LIN {X 0.200,Y -475.313,Z 1141.533,A 0.000,B 0.000,C 90.000,E1 275.853} C_DIS
LIN {X -0.137,Y -474.500,Z 1141.530,A 0.000,B 0.000,C 90.000,E1 275.391} C_DIS
LIN {X -0.046,Y -473.245,Z 1141.527,A 0.000,B 0.000,C 90.000,E1 274.878} C_DIS
LIN {X 0.081,Y -471.579,Z 1141.524,A 0.000,B 0.000,C 90.000,E1 274.359} C_DIS
LIN {X 0.199,Y -469.321,Z 1141.521,A 0.000,B 0.000,C 90.000,E1 273.841} C_DIS
LIN {X 0.000,Y -468.016,Z 1141.520,A 0.000,B 0.000,C 90.000,E1 273.612} C_DIS
LIN {X 0.090,Y -464.739,Z 1141.517,A 0.000,B 0.000,C 90.000,E1 273.094} C_DIS
LIN {X -0.113,Y -462.816,Z 1141.516,A 0.000,B 0.000,C 90.000,E1 272.865} C_DIS
LIN {X -0.071,Y -458.078,Z 1141.513,A 0.000,B 0.000,C 90.000,E1 272.350} C_DIS
LIN {X 0.192,Y -455.207,Z 1141.512,A 0.000,B 0.000,C 90.000,E1 272.064} C_DIS
LIN {X 0.157,Y -448.955,Z 1141.509,A 0.000,B 0.000,C 90.000,E1 271.604} C_DIS
LIN {X -0.185,Y -442.338,Z 1141.507,A 0.000,B 0.000,C 90.000,E1 271.260} C_DIS
LIN {X -0.038,Y -435.436,Z 1141.505,A 0.000,B 0.000,C 90.000,E1 270.917} C_DIS
LIN {X 0.066,Y -428.431,Z 1141.504,A 0.000,B 0.000,C 90.000,E1 270.630} C_DIS
LIN {X 0.073,Y -421.301,Z 1141.502,A 0.000,B 0.000,C 90.000,E1 270.401} C_DIS
LIN {X -0.072,Y -414.046,Z 1141.501,A 0.000,B 0.000,C 90.000,E1 270.229} C_DIS
LIN {X -0.082,Y -402.883,Z 1141.500,A 0.000,B 0.000,C 90.000,E1 270.000} C_DIS
LIN {X -0.091,Y -391.480,Z 1141.499,A 0.000,B 0.000,C 90.000,E1 269.828} C_DIS
LIN {X -0.150,Y -380.857,Z 1141.499,A 0.000,B 0.000,C 90.000,E1 269.771} C_DIS
LIN {X 0.176,Y -377.810,Z 1141.499,A 0.000,B 0.000,C 90.000,E1 269.714} C_DIS
LIN {X 0.059,Y -181.500,Z 1141.499,A 0.000,B 0.000,C 90.000,E1 269.714} C_DIS
LIN {X 0.062,Y -180.907,Z 1141.475,A 0.000,B 0.000,C 90.000,E1 265.469} C_DIS
LIN {X -0.062,Y -180.745,Z 1141.470,A 0.000,B 0.000,C 90.000,E1 264.666} C_DIS
LIN {X 0.007,Y -178.837,Z 1141.442,A 0.000,B 0.000,C 90.000,E1 259.577} C_DIS
LIN {X -0.096,Y -175.880,Z 1141.414,A 0.000,B 0.000,C 90.000,E1 254.519} C_DIS
LIN {X 0.010,Y -174.542,Z 1141.404,A 0.000,B 0.000,C 90.000,E1 252.779} C_DIS
LIN {X 0.103,Y -171.527,Z 1141.380,A 0.000,B 0.000,C 90.000,E1 248.465} C_DIS
LIN {X 0.089,Y -167.753,Z 1141.357,A 0.000,B 0.000,C 90.000,E1 244.152} C_DIS
LIN {X 0.026,Y -166.456,Z 1141.347,A 0.000,B 0.000,C 90.000,E1 242.436} C_DIS
LIN {X 0.017,Y -163.172,Z 1141.328,A 0.000,B 0.000,C 90.000,E1 238.948} C_DIS
LIN {X 0.066,Y -161.131,Z 1141.313,A 0.000,B 0.000,C 90.000,E1 236.294} C_DIS
LIN {X -0.032,Y -157.153,Z 1141.288,A 0.000,B 0.000,C 90.000,E1 231.904} C_DIS
LIN {X -0.009,Y -155.885,Z 1141.278,A 0.000,B 0.000,C 90.000,E1 230.114} C_DIS
LIN {X -0.050,Y -152.135,Z 1141.254,A 0.000,B 0.000,C 90.000,E1 225.648} C_DIS
LIN {X -0.030,Y -150.385,Z 1141.238,A 0.000,B 0.000,C 90.000,E1 222.933} C_DIS
LIN {X -0.005,Y -147.117,Z 1141.213,A 0.000,B 0.000,C 90.000,E1 218.382} C_DIS
LIN {X -0.015,Y -145.682,Z 1141.198,A 0.000,B 0.000,C 90.000,E1 215.644} C_DIS
LIN {X -0.017,Y -143.065,Z 1141.172,A 0.000,B 0.000,C 90.000,E1 211.052} C_DIS
LIN {X 0.041,Y -141.686,Z 1141.152,A 0.000,B 0.000,C 90.000,E1 207.334} C_DIS
LIN {X 0.019,Y -139.459,Z 1141.116,A 0.000,B 0.000,C 90.000,E1 200.844} C_DIS
LIN {X 0.069,Y -139.193,Z 1141.105,A 0.000,B 0.000,C 90.000,E1 198.960} C_DIS
LIN {X -0.044,Y -138.325,Z 1141.054,A 0.000,B 0.000,C 90.000,E1 189.670} C_DIS
LIN {X -0.039,Y -139.453,Z 1141.007,A 0.000,B 0.000,C 90.000,E1 181.260} C_DIS
LIN {X 0.041,Y -141.000,Z 1140.976,A 0.000,B 0.000,C 90.000,E1 175.641} C_DIS
LIN {X -0.009,Y -142.755,Z 1140.955,A 0.000,B 0.000,C 90.000,E1 171.951} C_DIS
LIN {X -0.054,Y -145.157,Z 1140.930,A 0.000,B 0.000,C 90.000,E1 167.353} C_DIS
LIN {X -0.061,Y -147.779,Z 1140.909,A 0.000,B 0.000,C 90.000,E1 163.685} C_DIS
LIN {X 0.019,Y -150.457,Z 1140.889,A 0.000,B 0.000,C 90.000,E1 160.007} C_DIS
LIN {X -0.048,Y -153.906,Z 1140.869,A 0.000,B 0.000,C 90.000,E1 156.410} C_DIS
LIN {X 0.017,Y -157.316,Z 1140.849,A 0.000,B 0.000,C 90.000,E1 152.794} C_DIS
LIN {X -0.036,Y -161.504,Z 1140.829,A 0.000,B 0.000,C 90.000,E1 149.253} C_DIS
LIN {X -0.020,Y -165.703,Z 1140.810,A 0.000,B 0.000,C 90.000,E1 145.722} C_DIS
LIN {X 0.106,Y -170.649,Z 1140.790,A 0.000,B 0.000,C 90.000,E1 142.190} C_DIS
LIN {X 0.018,Y -175.524,Z 1140.771,A 0.000,B 0.000,C 90.000,E1 138.771} C_DIS
LIN {X 0.012,Y -181.144,Z 1140.752,A 0.000,B 0.000,C 90.000,E1 135.364} C_DIS
LIN {X 0.010,Y -186.596,Z 1140.733,A 0.000,B 0.000,C 90.000,E1 132.000} C_DIS
LIN {X 0.080,Y -191.206,Z 1140.719,A 0.000,B 0.000,C 90.000,E1 129.483} C_DIS
LIN {X 0.004,Y -197.018,Z 1140.701,A 0.000,B 0.000,C 90.000,E1 126.217} C_DIS
LIN {X -0.072,Y -201.191,Z 1140.689,A 0.000,B 0.000,C 90.000,E1 124.119} C_DIS
LIN {X 0.092,Y -310.929,Z 1140.689,A 0.000,B 0.000,C 90.000,E1 124.072} C_DIS
LIN {X 0.092,Y -315.579,Z 1140.688,A 0.000,B 0.000,C 90.000,E1 123.913} C_DIS
LIN {X -0.033,Y -317.772,Z 1140.688,A 0.000,B 0.000,C 90.000,E1 123.785} C_DIS
LIN {X -0.005,Y -321.647,Z 1140.685,A 0.000,B 0.000,C 90.000,E1 123.372} C_DIS
LIN {X -0.032,Y -323.552,Z 1140.684,A 0.000,B 0.000,C 90.000,E1 123.086} C_DIS
LIN {X -0.060,Y -325.048,Z 1140.682,A 0.000,B 0.000,C 90.000,E1 122.801} C_DIS
LIN {X -0.046,Y -328.621,Z 1140.677,A 0.000,B 0.000,C 90.000,E1 121.848} C_DIS
LIN {X -0.027,Y -339.698,Z 1140.661,A 0.000,B 0.000,C 90.000,E1 119.027} C_DIS
LIN {X 0.170,Y -352.167,Z 1140.646,A 0.000,B 0.000,C 90.000,E1 116.232} C_DIS
LIN {X -0.081,Y -366.144,Z 1140.631,A 0.000,B 0.000,C 90.000,E1 113.567} C_DIS
LIN {X -0.161,Y -379.928,Z 1140.618,A 0.000,B 0.000,C 90.000,E1 111.227} C_DIS
LIN {X -0.023,Y -395.095,Z 1140.605,A 0.000,B 0.000,C 90.000,E1 108.906} C_DIS
LIN {X -0.141,Y -411.753,Z 1140.593,A 0.000,B 0.000,C 90.000,E1 106.677} C_DIS
LIN {X -0.085,Y -430.020,Z 1140.580,A 0.000,B 0.000,C 90.000,E1 104.481} C_DIS
LIN {X 0.106,Y -449.754,Z 1140.569,A 0.000,B 0.000,C 90.000,E1 102.355} C_DIS
LIN {X 0.080,Y -467.535,Z 1140.559,A 0.000,B 0.000,C 90.000,E1 100.658} C_DIS
LIN {X 0.008,Y -469.919,Z 1140.558,A 0.000,B 0.000,C 90.000,E1 100.433} C_DIS
LIN {X -0.067,Y -471.794,Z 1140.557,A 0.000,B 0.000,C 90.000,E1 100.197} C_DIS
LIN {X -0.143,Y -473.215,Z 1140.555,A 0.000,B 0.000,C 90.000,E1 99.962} C_DIS
LIN {X -0.037,Y -475.103,Z 1140.552,A 0.000,B 0.000,C 90.000,E1 99.443} C_DIS
LIN {X 0.157,Y -475.883,Z 1140.550,A 0.000,B 0.000,C 90.000,E1 98.916} C_DIS
LIN {X -0.184,Y -475.689,Z 1140.547,A 0.000,B 0.000,C 90.000,E1 98.454} C_DIS
LIN {X -0.047,Y -474.497,Z 1140.544,A 0.000,B 0.000,C 90.000,E1 97.936} C_DIS
LIN {X -0.182,Y -473.472,Z 1140.543,A 0.000,B 0.000,C 90.000,E1 97.701} C_DIS
LIN {X 0.151,Y -472.094,Z 1140.541,A 0.000,B 0.000,C 90.000,E1 97.409} C_DIS
LIN {X 0.048,Y -457.591,Z 1140.530,A 0.000,B 0.000,C 90.000,E1 95.391} C_DIS
LIN {X 0.126,Y -438.390,Z 1140.514,A 0.000,B 0.000,C 90.000,E1 92.522} C_DIS
LIN {X 0.138,Y -419.215,Z 1140.496,A 0.000,B 0.000,C 90.000,E1 89.312} C_DIS
LIN {X -0.010,Y -408.971,Z 1140.486,A 0.000,B 0.000,C 90.000,E1 87.421} C_DIS
LIN {X 0.054,Y -398.485,Z 1140.475,A 0.000,B 0.000,C 90.000,E1 85.469} C_DIS
LIN {X 0.018,Y -385.098,Z 1140.461,A 0.000,B 0.000,C 90.000,E1 82.932} C_DIS
LIN {X 0.082,Y -376.107,Z 1140.451,A 0.000,B 0.000,C 90.000,E1 81.197} C_DIS
LIN {X 0.036,Y -366.859,Z 1140.441,A 0.000,B 0.000,C 90.000,E1 79.454} C_DIS
LIN {X -0.074,Y -358.902,Z 1140.433,A 0.000,B 0.000,C 90.000,E1 77.993} C_DIS
LIN {X -0.002,Y -347.398,Z 1140.422,A 0.000,B 0.000,C 90.000,E1 75.880} C_DIS
LIN {X -0.026,Y -334.287,Z 1140.408,A 0.000,B 0.000,C 90.000,E1 73.433} C_DIS
LIN {X -0.001,Y -320.080,Z 1140.392,A 0.000,B 0.000,C 90.000,E1 70.604} C_DIS
LIN {X 0.053,Y -303.837,Z 1140.373,A 0.000,B 0.000,C 90.000,E1 67.050} C_DIS
LIN {X 0.038,Y -291.318,Z 1140.356,A 0.000,B 0.000,C 90.000,E1 64.076} C_DIS
LIN {X -0.058,Y -279.221,Z 1140.339,A 0.000,B 0.000,C 90.000,E1 61.051} C_DIS
LIN {X 0.049,Y -267.755,Z 1140.322,A 0.000,B 0.000,C 90.000,E1 57.916} C_DIS
LIN {X -0.102,Y -256.802,Z 1140.304,A 0.000,B 0.000,C 90.000,E1 54.769} C_DIS
LIN {X 0.031,Y -245.381,Z 1140.284,A 0.000,B 0.000,C 90.000,E1 51.126} C_DIS
LIN {X -0.112,Y -235.027,Z 1140.264,A 0.000,B 0.000,C 90.000,E1 47.472} C_DIS
LIN {X 0.030,Y -227.285,Z 1140.247,A 0.000,B 0.000,C 90.000,E1 44.433} C_DIS
LIN {X -0.012,Y -218.155,Z 1140.226,A 0.000,B 0.000,C 90.000,E1 40.620} C_DIS
LIN {X -0.066,Y -211.276,Z 1140.208,A 0.000,B 0.000,C 90.000,E1 37.523} C_DIS
LIN {X 0.079,Y -204.769,Z 1140.191,A 0.000,B 0.000,C 90.000,E1 34.326} C_DIS
LIN {X 0.015,Y -197.461,Z 1140.169,A 0.000,B 0.000,C 90.000,E1 30.335} C_DIS
LIN {X 0.028,Y -192.220,Z 1140.151,A 0.000,B 0.000,C 90.000,E1 27.078} C_DIS
LIN {X 0.055,Y -186.581,Z 1140.128,A 0.000,B 0.000,C 90.000,E1 22.950} C_DIS
LIN {X 0.058,Y -181.865,Z 1140.104,A 0.000,B 0.000,C 90.000,E1 18.779} C_DIS
LIN {X -0.023,Y -178.162,Z 1140.081,A 0.000,B 0.000,C 90.000,E1 14.592} C_DIS
LIN {X -0.047,Y -175.079,Z 1140.053,A 0.000,B 0.000,C 90.000,E1 9.500} C_DIS
LIN {X 0.015,Y -173.270,Z 1140.005,A 0.000,B 0.000,C 90.000,E1 0.917} C_DIS
LIN {X 0.050,Y -174.989,Z 1139.964,A 0.000,B 0.000,C 90.000,E1 353.514} C_DIS
LIN {X 0.006,Y -177.963,Z 1139.936,A 0.000,B 0.000,C 90.000,E1 348.409} C_DIS
LIN {X 0.056,Y -181.448,Z 1139.912,A 0.000,B 0.000,C 90.000,E1 344.157} C_DIS
LIN {X -0.110,Y -185.852,Z 1139.889,A 0.000,B 0.000,C 90.000,E1 340.007} C_DIS
LIN {X 0.074,Y -191.032,Z 1139.866,A 0.000,B 0.000,C 90.000,E1 335.793} C_DIS
LIN {X -0.045,Y -195.878,Z 1139.847,A 0.000,B 0.000,C 90.000,E1 332.538} C_DIS
LIN {X -0.043,Y -201.277,Z 1139.829,A 0.000,B 0.000,C 90.000,E1 329.282} C_DIS
LIN {X -0.121,Y -207.264,Z 1139.811,A 0.000,B 0.000,C 90.000,E1 326.087} C_DIS
LIN {X -0.032,Y -214.122,Z 1139.794,A 0.000,B 0.000,C 90.000,E1 322.889} C_DIS
LIN {X -0.049,Y -222.780,Z 1139.774,A 0.000,B 0.000,C 90.000,E1 319.380} C_DIS
LIN {X 0.034,Y -231.481,Z 1139.757,A 0.000,B 0.000,C 90.000,E1 316.296} C_DIS
LIN {X 0.001,Y -241.200,Z 1139.741,A 0.000,B 0.000,C 90.000,E1 313.299} C_DIS
LIN {X -0.106,Y -252.087,Z 1139.724,A 0.000,B 0.000,C 90.000,E1 310.378} C_DIS
LIN {X 0.139,Y -264.307,Z 1139.708,A 0.000,B 0.000,C 90.000,E1 307.443} C_DIS
LIN {X -0.053,Y -279.632,Z 1139.691,A 0.000,B 0.000,C 90.000,E1 304.326} C_DIS
LIN {X -0.018,Y -292.655,Z 1139.677,A 0.000,B 0.000,C 90.000,E1 301.926} C_DIS
LIN {X -0.124,Y -308.904,Z 1139.663,A 0.000,B 0.000,C 90.000,E1 299.283} C_DIS
LIN {X 0.042,Y -326.808,Z 1139.648,A 0.000,B 0.000,C 90.000,E1 296.668} C_DIS
LIN {X 0.124,Y -341.553,Z 1139.638,A 0.000,B 0.000,C 90.000,E1 294.771} C_DIS
LIN {X 0.091,Y -354.713,Z 1139.629,A 0.000,B 0.000,C 90.000,E1 293.259} C_DIS
LIN {X 0.010,Y -368.110,Z 1139.622,A 0.000,B 0.000,C 90.000,E1 291.897} C_DIS
LIN {X -0.061,Y -392.786,Z 1139.609,A 0.000,B 0.000,C 90.000,E1 289.631} C_DIS
LIN {X -0.033,Y -403.534,Z 1139.604,A 0.000,B 0.000,C 90.000,E1 288.652} C_DIS
LIN {X 0.210,Y -411.431,Z 1139.599,A 0.000,B 0.000,C 90.000,E1 287.873} C_DIS
LIN {X 0.215,Y -421.680,Z 1139.594,A 0.000,B 0.000,C 90.000,E1 286.858} C_DIS
LIN {X 0.218,Y -429.215,Z 1139.589,A 0.000,B 0.000,C 90.000,E1 286.079} C_DIS
LIN {X 0.086,Y -436.426,Z 1139.585,A 0.000,B 0.000,C 90.000,E1 285.300} C_DIS
LIN {X -0.180,Y -443.169,Z 1139.581,A 0.000,B 0.000,C 90.000,E1 284.537} C_DIS
LIN {X 0.056,Y -449.195,Z 1139.576,A 0.000,B 0.000,C 90.000,E1 283.716} C_DIS
LIN {X 0.011,Y -454.502,Z 1139.572,A 0.000,B 0.000,C 90.000,E1 282.939} C_DIS
LIN {X -0.091,Y -459.121,Z 1139.568,A 0.000,B 0.000,C 90.000,E1 282.175} C_DIS
LIN {X -0.252,Y -463.156,Z 1139.563,A 0.000,B 0.000,C 90.000,E1 281.422} C_DIS
LIN {X 0.020,Y -467.739,Z 1139.558,A 0.000,B 0.000,C 90.000,E1 280.366} C_DIS
LIN {X 0.093,Y -469.729,Z 1139.555,A 0.000,B 0.000,C 90.000,E1 279.849} C_DIS
LIN {X -0.209,Y -471.485,Z 1139.552,A 0.000,B 0.000,C 90.000,E1 279.378} C_DIS
LIN {X -0.115,Y -473.007,Z 1139.549,A 0.000,B 0.000,C 90.000,E1 278.859} C_DIS
LIN {X -0.005,Y -474.223,Z 1139.546,A 0.000,B 0.000,C 90.000,E1 278.341} C_DIS
LIN {X 0.180,Y -475.168,Z 1139.544,A 0.000,B 0.000,C 90.000,E1 277.814} C_DIS
LIN {X -0.164,Y -475.768,Z 1139.541,A 0.000,B 0.000,C 90.000,E1 277.352} C_DIS
LIN {X -0.032,Y -476.050,Z 1139.538,A 0.000,B 0.000,C 90.000,E1 276.834} C_DIS
LIN {X 0.105,Y -475.977,Z 1139.535,A 0.000,B 0.000,C 90.000,E1 276.315} C_DIS
LIN {X 0.243,Y -475.515,Z 1139.532,A 0.000,B 0.000,C 90.000,E1 275.796} C_DIS
LIN {X -0.094,Y -474.683,Z 1139.530,A 0.000,B 0.000,C 90.000,E1 275.334} C_DIS
LIN {X -0.002,Y -473.432,Z 1139.527,A 0.000,B 0.000,C 90.000,E1 274.821} C_DIS
LIN {X 0.128,Y -471.721,Z 1139.524,A 0.000,B 0.000,C 90.000,E1 274.302} C_DIS
LIN {X -0.223,Y -469.455,Z 1139.521,A 0.000,B 0.000,C 90.000,E1 273.841} C_DIS
LIN {X -0.150,Y -466.592,Z 1139.518,A 0.000,B 0.000,C 90.000,E1 273.326} C_DIS
LIN {X -0.065,Y -462.911,Z 1139.516,A 0.000,B 0.000,C 90.000,E1 272.808} C_DIS
LIN {X -0.023,Y -458.133,Z 1139.513,A 0.000,B 0.000,C 90.000,E1 272.293} C_DIS
LIN {X -0.206,Y -455.209,Z 1139.511,A 0.000,B 0.000,C 90.000,E1 272.064} C_DIS
LIN {X -0.213,Y -448.901,Z 1139.509,A 0.000,B 0.000,C 90.000,E1 271.604} C_DIS
LIN {X -0.091,Y -442.192,Z 1139.507,A 0.000,B 0.000,C 90.000,E1 271.203} C_DIS
LIN {X 0.068,Y -435.279,Z 1139.505,A 0.000,B 0.000,C 90.000,E1 270.859} C_DIS
LIN {X 0.194,Y -428.312,Z 1139.503,A 0.000,B 0.000,C 90.000,E1 270.573} C_DIS
LIN {X -0.207,Y -421.182,Z 1139.502,A 0.000,B 0.000,C 90.000,E1 270.401} C_DIS
LIN {X 0.081,Y -413.850,Z 1139.501,A 0.000,B 0.000,C 90.000,E1 270.172} C_DIS
LIN {X 0.084,Y -402.501,Z 1139.500,A 0.000,B 0.000,C 90.000,E1 269.943} C_DIS
LIN {X 0.059,Y -394.923,Z 1139.499,A 0.000,B 0.000,C 90.000,E1 269.828} C_DIS
LIN {X -0.055,Y -388.034,Z 1139.499,A 0.000,B 0.000,C 90.000,E1 269.771} C_DIS
LIN {X 0.056,Y -378.077,Z 1139.498,A 0.000,B 0.000,C 90.000,E1 269.714} C_DIS
LIN {X 0.001,Y -181.494,Z 1139.498,A 0.000,B 0.000,C 90.000,E1 269.714} C_DIS
LIN {X -0.020,Y -180.907,Z 1139.475,A 0.000,B 0.000,C 90.000,E1 265.469} C_DIS
LIN {X 0.037,Y -180.733,Z 1139.470,A 0.000,B 0.000,C 90.000,E1 264.609} C_DIS
LIN {X -0.042,Y -178.823,Z 1139.442,A 0.000,B 0.000,C 90.000,E1 259.567} C_DIS
LIN {X 0.040,Y -175.868,Z 1139.414,A 0.000,B 0.000,C 90.000,E1 254.448} C_DIS
LIN {X 0.034,Y -173.838,Z 1139.399,A 0.000,B 0.000,C 90.000,E1 251.891} C_DIS
LIN {X 0.023,Y -171.505,Z 1139.380,A 0.000,B 0.000,C 90.000,E1 248.465} C_DIS
LIN {X 0.010,Y -167.733,Z 1139.356,A 0.000,B 0.000,C 90.000,E1 244.152} C_DIS
LIN {X 0.026,Y -166.430,Z 1139.347,A 0.000,B 0.000,C 90.000,E1 242.410} C_DIS
LIN {X -0.060,Y -163.150,Z 1139.327,A 0.000,B 0.000,C 90.000,E1 238.948} C_DIS
LIN {X -0.011,Y -161.105,Z 1139.313,A 0.000,B 0.000,C 90.000,E1 236.294} C_DIS
LIN {X -0.027,Y -157.833,Z 1139.293,A 0.000,B 0.000,C 90.000,E1 232.763} C_DIS
LIN {X 0.036,Y -155.865,Z 1139.278,A 0.000,B 0.000,C 90.000,E1 230.070} C_DIS
LIN {X 0.091,Y -152.115,Z 1139.253,A 0.000,B 0.000,C 90.000,E1 225.567} C_DIS
LIN {X -0.001,Y -150.366,Z 1139.238,A 0.000,B 0.000,C 90.000,E1 222.894} C_DIS
LIN {X 0.038,Y -147.101,Z 1139.213,A 0.000,B 0.000,C 90.000,E1 218.338} C_DIS
LIN {X 0.031,Y -145.669,Z 1139.198,A 0.000,B 0.000,C 90.000,E1 215.598} C_DIS
LIN {X 0.035,Y -143.051,Z 1139.172,A 0.000,B 0.000,C 90.000,E1 211.003} C_DIS
LIN {X -0.030,Y -141.674,Z 1139.152,A 0.000,B 0.000,C 90.000,E1 207.334} C_DIS
LIN {X 0.079,Y -139.454,Z 1139.116,A 0.000,B 0.000,C 90.000,E1 200.791} C_DIS
LIN {X 0.000,Y -139.188,Z 1139.105,A 0.000,B 0.000,C 90.000,E1 198.960} C_DIS
LIN {X 0.023,Y -138.323,Z 1139.053,A 0.000,B 0.000,C 90.000,E1 189.613} C_DIS
LIN {X 0.030,Y -139.458,Z 1139.007,A 0.000,B 0.000,C 90.000,E1 181.203} C_DIS
LIN {X -0.029,Y -141.012,Z 1138.976,A 0.000,B 0.000,C 90.000,E1 175.641} C_DIS
LIN {X 0.061,Y -142.766,Z 1138.955,A 0.000,B 0.000,C 90.000,E1 171.894} C_DIS
LIN {X 0.016,Y -145.175,Z 1138.929,A 0.000,B 0.000,C 90.000,E1 167.297} C_DIS
LIN {X 0.050,Y -147.796,Z 1138.909,A 0.000,B 0.000,C 90.000,E1 163.614} C_DIS
LIN {X -0.055,Y -150.480,Z 1138.889,A 0.000,B 0.000,C 90.000,E1 160.007} C_DIS
LIN {X 0.019,Y -153.935,Z 1138.869,A 0.000,B 0.000,C 90.000,E1 156.357} C_DIS
LIN {X 0.082,Y -157.346,Z 1138.849,A 0.000,B 0.000,C 90.000,E1 152.743} C_DIS
LIN {X 0.026,Y -161.540,Z 1138.829,A 0.000,B 0.000,C 90.000,E1 149.203} C_DIS
LIN {X 0.039,Y -165.738,Z 1138.809,A 0.000,B 0.000,C 90.000,E1 145.674} C_DIS
LIN {X 0.026,Y -170.691,Z 1138.790,A 0.000,B 0.000,C 90.000,E1 142.190} C_DIS
LIN {X -0.062,Y -175.564,Z 1138.771,A 0.000,B 0.000,C 90.000,E1 138.771} C_DIS
LIN {X 0.057,Y -181.182,Z 1138.752,A 0.000,B 0.000,C 90.000,E1 135.324} C_DIS
LIN {X -0.074,Y -186.642,Z 1138.733,A 0.000,B 0.000,C 90.000,E1 132.000} C_DIS
LIN {X -0.005,Y -191.248,Z 1138.719,A 0.000,B 0.000,C 90.000,E1 129.483} C_DIS
LIN {X -0.082,Y -197.066,Z 1138.701,A 0.000,B 0.000,C 90.000,E1 126.217} C_DIS
LIN {X -0.010,Y -201.161,Z 1138.690,A 0.000,B 0.000,C 90.000,E1 124.119} C_DIS
LIN {X -0.074,Y -310.690,Z 1138.689,A 0.000,B 0.000,C 90.000,E1 124.119} C_DIS
LIN {X 0.066,Y -315.833,Z 1138.688,A 0.000,B 0.000,C 90.000,E1 123.913} C_DIS
LIN {X -0.171,Y -318.170,Z 1138.688,A 0.000,B 0.000,C 90.000,E1 123.785} C_DIS
LIN {X 0.172,Y -322.022,Z 1138.685,A 0.000,B 0.000,C 90.000,E1 123.293} C_DIS
LIN {X -0.104,Y -323.897,Z 1138.683,A 0.000,B 0.000,C 90.000,E1 123.038} C_DIS
LIN {X 0.068,Y -325.366,Z 1138.682,A 0.000,B 0.000,C 90.000,E1 122.704} C_DIS
LIN {X -0.132,Y -338.678,Z 1138.663,A 0.000,B 0.000,C 90.000,E1 119.283} C_DIS
LIN {X 0.025,Y -351.027,Z 1138.647,A 0.000,B 0.000,C 90.000,E1 116.488} C_DIS
LIN {X 0.078,Y -364.867,Z 1138.632,A 0.000,B 0.000,C 90.000,E1 113.770} C_DIS
LIN {X 0.120,Y -378.524,Z 1138.619,A 0.000,B 0.000,C 90.000,E1 111.408} C_DIS
LIN {X -0.140,Y -393.553,Z 1138.606,A 0.000,B 0.000,C 90.000,E1 109.141} C_DIS
LIN {X 0.087,Y -410.062,Z 1138.594,A 0.000,B 0.000,C 90.000,E1 106.858} C_DIS
LIN {X 0.112,Y -428.168,Z 1138.582,A 0.000,B 0.000,C 90.000,E1 104.662} C_DIS
LIN {X -0.214,Y -447.792,Z 1138.570,A 0.000,B 0.000,C 90.000,E1 102.591} C_DIS
LIN {X 0.091,Y -468.110,Z 1138.559,A 0.000,B 0.000,C 90.000,E1 100.602} C_DIS
LIN {X 0.110,Y -470.350,Z 1138.558,A 0.000,B 0.000,C 90.000,E1 100.366} C_DIS
LIN {X -0.122,Y -472.163,Z 1138.556,A 0.000,B 0.000,C 90.000,E1 100.141} C_DIS
LIN {X 0.196,Y -473.524,Z 1138.555,A 0.000,B 0.000,C 90.000,E1 99.849} C_DIS
LIN {X -0.084,Y -475.233,Z 1138.552,A 0.000,B 0.000,C 90.000,E1 99.378} C_DIS
LIN {X 0.034,Y -475.869,Z 1138.549,A 0.000,B 0.000,C 90.000,E1 98.859} C_DIS
LIN {X 0.167,Y -475.536,Z 1138.547,A 0.000,B 0.000,C 90.000,E1 98.341} C_DIS
LIN {X -0.102,Y -474.189,Z 1138.544,A 0.000,B 0.000,C 90.000,E1 97.871} C_DIS
LIN {X 0.168,Y -473.070,Z 1138.542,A 0.000,B 0.000,C 90.000,E1 97.587} C_DIS
LIN {X 0.030,Y -471.574,Z 1138.541,A 0.000,B 0.000,C 90.000,E1 97.352} C_DIS
LIN {X 0.145,Y -455.223,Z 1138.528,A 0.000,B 0.000,C 90.000,E1 95.049} C_DIS
LIN {X -0.183,Y -439.529,Z 1138.515,A 0.000,B 0.000,C 90.000,E1 92.751} C_DIS
LIN {X 0.178,Y -421.764,Z 1138.499,A 0.000,B 0.000,C 90.000,E1 89.771} C_DIS
LIN {X -0.165,Y -408.479,Z 1138.485,A 0.000,B 0.000,C 90.000,E1 87.364} C_DIS
LIN {X -0.108,Y -397.980,Z 1138.474,A 0.000,B 0.000,C 90.000,E1 85.412} C_DIS
LIN {X -0.153,Y -384.603,Z 1138.460,A 0.000,B 0.000,C 90.000,E1 82.875} C_DIS
LIN {X -0.096,Y -375.592,Z 1138.451,A 0.000,B 0.000,C 90.000,E1 81.141} C_DIS
LIN {X -0.148,Y -366.316,Z 1138.441,A 0.000,B 0.000,C 90.000,E1 79.398} C_DIS
LIN {X 0.086,Y -358.335,Z 1138.433,A 0.000,B 0.000,C 90.000,E1 77.881} C_DIS
LIN {X -0.117,Y -346.817,Z 1138.421,A 0.000,B 0.000,C 90.000,E1 75.811} C_DIS
LIN {X 0.085,Y -333.720,Z 1138.407,A 0.000,B 0.000,C 90.000,E1 73.323} C_DIS
LIN {X 0.080,Y -319.500,Z 1138.392,A 0.000,B 0.000,C 90.000,E1 70.496} C_DIS
LIN {X -0.063,Y -303.309,Z 1138.372,A 0.000,B 0.000,C 90.000,E1 66.975} C_DIS
LIN {X 0.053,Y -290.796,Z 1138.355,A 0.000,B 0.000,C 90.000,E1 63.973} C_DIS
LIN {X 0.066,Y -278.715,Z 1138.339,A 0.000,B 0.000,C 90.000,E1 60.923} C_DIS
LIN {X 0.151,Y -267.269,Z 1138.321,A 0.000,B 0.000,C 90.000,E1 57.788} C_DIS
LIN {X -0.021,Y -256.318,Z 1138.304,A 0.000,B 0.000,C 90.000,E1 54.642} C_DIS
LIN {X 0.041,Y -245.979,Z 1138.286,A 0.000,B 0.000,C 90.000,E1 51.376} C_DIS
LIN {X -0.032,Y -236.536,Z 1138.267,A 0.000,B 0.000,C 90.000,E1 48.081} C_DIS
LIN {X -0.012,Y -228.708,Z 1138.250,A 0.000,B 0.000,C 90.000,E1 45.081} C_DIS
LIN {X -0.025,Y -219.457,Z 1138.229,A 0.000,B 0.000,C 90.000,E1 41.272} C_DIS
LIN {X -0.052,Y -212.462,Z 1138.212,A 0.000,B 0.000,C 90.000,E1 38.177} C_DIS
LIN {X 0.071,Y -204.260,Z 1138.190,A 0.000,B 0.000,C 90.000,E1 34.199} C_DIS
LIN {X -0.004,Y -196.963,Z 1138.168,A 0.000,B 0.000,C 90.000,E1 30.207} C_DIS
LIN {X -0.002,Y -191.740,Z 1138.150,A 0.000,B 0.000,C 90.000,E1 26.950} C_DIS
LIN {X 0.011,Y -186.124,Z 1138.127,A 0.000,B 0.000,C 90.000,E1 22.823} C_DIS
LIN {X -0.059,Y -181.433,Z 1138.104,A 0.000,B 0.000,C 90.000,E1 18.671} C_DIS
LIN {X 0.029,Y -177.741,Z 1138.080,A 0.000,B 0.000,C 90.000,E1 14.426} C_DIS
LIN {X 0.027,Y -174.715,Z 1138.052,A 0.000,B 0.000,C 90.000,E1 9.321} C_DIS
LIN {X 0.000,Y -173.011,Z 1138.000,A 0.000,B 0.000,C 90.000,E1 360.000} C_DIS
LIN {X 0.071,Y -175.091,Z 1137.959,A 0.000,B 0.000,C 90.000,E1 352.648} C_DIS
LIN {X 0.100,Y -178.266,Z 1137.931,A 0.000,B 0.000,C 90.000,E1 347.521} C_DIS
LIN {X -0.011,Y -181.920,Z 1137.907,A 0.000,B 0.000,C 90.000,E1 343.323} C_DIS
LIN {X -0.041,Y -186.439,Z 1137.884,A 0.000,B 0.000,C 90.000,E1 339.135} C_DIS
LIN {X -0.007,Y -191.815,Z 1137.861,A 0.000,B 0.000,C 90.000,E1 334.973} C_DIS
LIN {X -0.019,Y -196.817,Z 1137.843,A 0.000,B 0.000,C 90.000,E1 331.691} C_DIS
LIN {X -0.064,Y -202.409,Z 1137.825,A 0.000,B 0.000,C 90.000,E1 328.456} C_DIS
LIN {X 0.006,Y -208.616,Z 1137.807,A 0.000,B 0.000,C 90.000,E1 325.229} C_DIS
LIN {X 0.008,Y -215.710,Z 1137.789,A 0.000,B 0.000,C 90.000,E1 322.065} C_DIS
LIN {X 0.079,Y -223.587,Z 1137.772,A 0.000,B 0.000,C 90.000,E1 318.933} C_DIS
LIN {X 0.018,Y -232.452,Z 1137.755,A 0.000,B 0.000,C 90.000,E1 315.891} C_DIS
LIN {X 0.010,Y -242.342,Z 1137.738,A 0.000,B 0.000,C 90.000,E1 312.894} C_DIS
LIN {X 0.123,Y -253.399,Z 1137.722,A 0.000,B 0.000,C 90.000,E1 309.930} C_DIS
LIN {X 0.041,Y -265.853,Z 1137.706,A 0.000,B 0.000,C 90.000,E1 307.076} C_DIS
LIN {X 0.124,Y -281.426,Z 1137.689,A 0.000,B 0.000,C 90.000,E1 303.913} C_DIS
LIN {X 0.044,Y -296.633,Z 1137.673,A 0.000,B 0.000,C 90.000,E1 301.209} C_DIS
LIN {X 0.006,Y -311.175,Z 1137.661,A 0.000,B 0.000,C 90.000,E1 298.899} C_DIS
LIN {X 0.095,Y -329.306,Z 1137.646,A 0.000,B 0.000,C 90.000,E1 296.309} C_DIS
LIN {X -0.057,Y -341.674,Z 1137.638,A 0.000,B 0.000,C 90.000,E1 294.771} C_DIS
LIN {X 0.044,Y -354.650,Z 1137.629,A 0.000,B 0.000,C 90.000,E1 293.259} C_DIS
LIN {X 0.023,Y -367.940,Z 1137.622,A 0.000,B 0.000,C 90.000,E1 291.897} C_DIS
LIN {X -0.176,Y -392.823,Z 1137.609,A 0.000,B 0.000,C 90.000,E1 289.631} C_DIS
LIN {X -0.119,Y -403.540,Z 1137.604,A 0.000,B 0.000,C 90.000,E1 288.652} C_DIS
LIN {X -0.001,Y -414.081,Z 1137.598,A 0.000,B 0.000,C 90.000,E1 287.638} C_DIS
LIN {X -0.057,Y -424.299,Z 1137.592,A 0.000,B 0.000,C 90.000,E1 286.622} C_DIS
LIN {X -0.100,Y -431.763,Z 1137.588,A 0.000,B 0.000,C 90.000,E1 285.843} C_DIS
LIN {X 0.178,Y -438.825,Z 1137.583,A 0.000,B 0.000,C 90.000,E1 285.009} C_DIS
LIN {X -0.056,Y -445.334,Z 1137.579,A 0.000,B 0.000,C 90.000,E1 284.245} C_DIS
LIN {X -0.135,Y -451.185,Z 1137.575,A 0.000,B 0.000,C 90.000,E1 283.467} C_DIS
LIN {X 0.177,Y -456.297,Z 1137.570,A 0.000,B 0.000,C 90.000,E1 282.647} C_DIS
LIN {X 0.088,Y -460.738,Z 1137.566,A 0.000,B 0.000,C 90.000,E1 281.883} C_DIS
LIN {X -0.050,Y -464.590,Z 1137.562,A 0.000,B 0.000,C 90.000,E1 281.130} C_DIS
LIN {X -0.070,Y -467.965,Z 1137.557,A 0.000,B 0.000,C 90.000,E1 280.366} C_DIS
LIN {X 0.168,Y -471.742,Z 1137.552,A 0.000,B 0.000,C 90.000,E1 279.321} C_DIS
LIN {X -0.201,Y -473.257,Z 1137.549,A 0.000,B 0.000,C 90.000,E1 278.859} C_DIS
LIN {X -0.091,Y -474.489,Z 1137.546,A 0.000,B 0.000,C 90.000,E1 278.341} C_DIS
LIN {X 0.096,Y -475.393,Z 1137.543,A 0.000,B 0.000,C 90.000,E1 277.814} C_DIS
LIN {X 0.225,Y -475.998,Z 1137.541,A 0.000,B 0.000,C 90.000,E1 277.296} C_DIS
LIN {X -0.113,Y -476.274,Z 1137.538,A 0.000,B 0.000,C 90.000,E1 276.834} C_DIS
LIN {X 0.024,Y -476.203,Z 1137.535,A 0.000,B 0.000,C 90.000,E1 276.315} C_DIS
LIN {X 0.164,Y -475.768,Z 1137.532,A 0.000,B 0.000,C 90.000,E1 275.796} C_DIS
LIN {X -0.172,Y -474.942,Z 1137.530,A 0.000,B 0.000,C 90.000,E1 275.334} C_DIS
LIN {X -0.077,Y -473.708,Z 1137.527,A 0.000,B 0.000,C 90.000,E1 274.821} C_DIS
LIN {X 0.053,Y -472.038,Z 1137.524,A 0.000,B 0.000,C 90.000,E1 274.302} C_DIS
LIN {X 0.173,Y -469.850,Z 1137.521,A 0.000,B 0.000,C 90.000,E1 273.784} C_DIS
LIN {X -0.220,Y -467.005,Z 1137.518,A 0.000,B 0.000,C 90.000,E1 273.326} C_DIS
LIN {X -0.133,Y -463.350,Z 1137.516,A 0.000,B 0.000,C 90.000,E1 272.808} C_DIS
LIN {X -0.088,Y -458.602,Z 1137.513,A 0.000,B 0.000,C 90.000,E1 272.293} C_DIS
LIN {X 0.189,Y -455.706,Z 1137.511,A 0.000,B 0.000,C 90.000,E1 272.007} C_DIS
LIN {X 0.169,Y -449.438,Z 1137.509,A 0.000,B 0.000,C 90.000,E1 271.547} C_DIS
LIN {X -0.164,Y -442.834,Z 1137.507,A 0.000,B 0.000,C 90.000,E1 271.203} C_DIS
LIN {X 0.002,Y -435.935,Z 1137.505,A 0.000,B 0.000,C 90.000,E1 270.859} C_DIS
LIN {X 0.120,Y -429.033,Z 1137.503,A 0.000,B 0.000,C 90.000,E1 270.573} C_DIS
LIN {X 0.109,Y -421.870,Z 1137.502,A 0.000,B 0.000,C 90.000,E1 270.344} C_DIS
LIN {X -0.045,Y -414.418,Z 1137.501,A 0.000,B 0.000,C 90.000,E1 270.172} C_DIS
LIN {X 0.054,Y -407.067,Z 1137.500,A 0.000,B 0.000,C 90.000,E1 270.000} C_DIS
LIN {X -0.053,Y -395.659,Z 1137.499,A 0.000,B 0.000,C 90.000,E1 269.828} C_DIS
LIN {X 0.044,Y -384.466,Z 1137.498,A 0.000,B 0.000,C 90.000,E1 269.714} C_DIS
LIN {X -0.067,Y -378.293,Z 1137.498,A 0.000,B 0.000,C 90.000,E1 269.714} C_DIS
LIN {X -0.059,Y -181.490,Z 1137.498,A 0.000,B 0.000,C 90.000,E1 269.714} C_DIS
LIN {X -0.085,Y -180.906,Z 1137.475,A 0.000,B 0.000,C 90.000,E1 265.469} C_DIS
LIN {X -0.028,Y -180.724,Z 1137.470,A 0.000,B 0.000,C 90.000,E1 264.609} C_DIS
LIN {X 0.070,Y -178.813,Z 1137.442,A 0.000,B 0.000,C 90.000,E1 259.511} C_DIS
LIN {X -0.024,Y -175.857,Z 1137.414,A 0.000,B 0.000,C 90.000,E1 254.448} C_DIS
LIN {X -0.042,Y -173.186,Z 1137.395,A 0.000,B 0.000,C 90.000,E1 251.040} C_DIS
LIN {X -0.040,Y -171.488,Z 1137.380,A 0.000,B 0.000,C 90.000,E1 248.465} C_DIS
LIN {X -0.052,Y -167.717,Z 1137.356,A 0.000,B 0.000,C 90.000,E1 244.152} C_DIS
LIN {X -0.036,Y -166.409,Z 1137.347,A 0.000,B 0.000,C 90.000,E1 242.410} C_DIS
LIN {X -0.038,Y -163.132,Z 1137.327,A 0.000,B 0.000,C 90.000,E1 238.918} C_DIS
LIN {X -0.071,Y -161.084,Z 1137.313,A 0.000,B 0.000,C 90.000,E1 236.294} C_DIS
LIN {X 0.038,Y -157.815,Z 1137.293,A 0.000,B 0.000,C 90.000,E1 232.718} C_DIS
LIN {X -0.024,Y -155.849,Z 1137.278,A 0.000,B 0.000,C 90.000,E1 230.070} C_DIS
LIN {X 0.033,Y -152.099,Z 1137.253,A 0.000,B 0.000,C 90.000,E1 225.567} C_DIS
LIN {X 0.051,Y -150.350,Z 1137.238,A 0.000,B 0.000,C 90.000,E1 222.852} C_DIS
LIN {X -0.020,Y -147.087,Z 1137.213,A 0.000,B 0.000,C 90.000,E1 218.338} C_DIS
LIN {X -0.025,Y -145.659,Z 1137.198,A 0.000,B 0.000,C 90.000,E1 215.598} C_DIS
LIN {X -0.022,Y -143.040,Z 1137.172,A 0.000,B 0.000,C 90.000,E1 211.003} C_DIS
LIN {X -0.021,Y -141.665,Z 1137.152,A 0.000,B 0.000,C 90.000,E1 207.308} C_DIS
LIN {X 0.023,Y -139.450,Z 1137.116,A 0.000,B 0.000,C 90.000,E1 200.791} C_DIS
LIN {X -0.055,Y -139.184,Z 1137.105,A 0.000,B 0.000,C 90.000,E1 198.960} C_DIS
LIN {X -0.032,Y -138.321,Z 1137.053,A 0.000,B 0.000,C 90.000,E1 189.613} C_DIS
LIN {X -0.025,Y -139.462,Z 1137.007,A 0.000,B 0.000,C 90.000,E1 181.203} C_DIS
LIN {X 0.055,Y -141.021,Z 1136.976,A 0.000,B 0.000,C 90.000,E1 175.584} C_DIS
LIN {X 0.009,Y -142.386,Z 1136.960,A 0.000,B 0.000,C 90.000,E1 172.818} C_DIS
LIN {X -0.070,Y -144.616,Z 1136.934,A 0.000,B 0.000,C 90.000,E1 168.229} C_DIS
LIN {X -0.008,Y -147.811,Z 1136.909,A 0.000,B 0.000,C 90.000,E1 163.614} C_DIS
LIN {X 0.079,Y -150.499,Z 1136.889,A 0.000,B 0.000,C 90.000,E1 159.934} C_DIS
LIN {X -0.041,Y -153.957,Z 1136.869,A 0.000,B 0.000,C 90.000,E1 156.357} C_DIS
LIN {X 0.021,Y -157.369,Z 1136.849,A 0.000,B 0.000,C 90.000,E1 152.743} C_DIS
LIN {X -0.036,Y -161.568,Z 1136.829,A 0.000,B 0.000,C 90.000,E1 149.203} C_DIS
LIN {X -0.025,Y -165.766,Z 1136.809,A 0.000,B 0.000,C 90.000,E1 145.674} C_DIS
LIN {X -0.038,Y -170.723,Z 1136.790,A 0.000,B 0.000,C 90.000,E1 142.190} C_DIS
LIN {X 0.005,Y -175.596,Z 1136.771,A 0.000,B 0.000,C 90.000,E1 138.728} C_DIS
LIN {X -0.008,Y -181.213,Z 1136.752,A 0.000,B 0.000,C 90.000,E1 135.324} C_DIS
LIN {X -0.016,Y -186.678,Z 1136.733,A 0.000,B 0.000,C 90.000,E1 131.962} C_DIS
LIN {X -0.073,Y -191.280,Z 1136.719,A 0.000,B 0.000,C 90.000,E1 129.483} C_DIS
LIN {X 0.008,Y -197.105,Z 1136.701,A 0.000,B 0.000,C 90.000,E1 126.171} C_DIS
LIN {X 0.091,Y -201.113,Z 1136.690,A 0.000,B 0.000,C 90.000,E1 124.119} C_DIS
LIN {X 0.105,Y -309.903,Z 1136.690,A 0.000,B 0.000,C 90.000,E1 124.119} C_DIS
LIN {X 0.004,Y -311.425,Z 1136.690,A 0.000,B 0.000,C 90.000,E1 124.119} C_DIS
LIN {X 0.081,Y -316.091,Z 1136.688,A 0.000,B 0.000,C 90.000,E1 123.913} C_DIS
LIN {X 0.160,Y -318.564,Z 1136.687,A 0.000,B 0.000,C 90.000,E1 123.706} C_DIS
LIN {X -0.086,Y -322.388,Z 1136.685,A 0.000,B 0.000,C 90.000,E1 123.293} C_DIS
LIN {X 0.003,Y -324.230,Z 1136.683,A 0.000,B 0.000,C 90.000,E1 122.959} C_DIS
LIN {X 0.094,Y -325.665,Z 1136.681,A 0.000,B 0.000,C 90.000,E1 122.625} C_DIS
LIN {X 0.054,Y -337.673,Z 1136.664,A 0.000,B 0.000,C 90.000,E1 119.489} C_DIS
LIN {X -0.115,Y -349.896,Z 1136.648,A 0.000,B 0.000,C 90.000,E1 116.744} C_DIS
LIN {X -0.104,Y -363.609,Z 1136.633,A 0.000,B 0.000,C 90.000,E1 114.027} C_DIS
LIN {X -0.096,Y -377.140,Z 1136.620,A 0.000,B 0.000,C 90.000,E1 111.663} C_DIS
LIN {X 0.109,Y -392.034,Z 1136.607,A 0.000,B 0.000,C 90.000,E1 109.322} C_DIS
LIN {X -0.085,Y -408.397,Z 1136.595,A 0.000,B 0.000,C 90.000,E1 107.094} C_DIS
LIN {X -0.112,Y -426.345,Z 1136.583,A 0.000,B 0.000,C 90.000,E1 104.898} C_DIS
LIN {X -0.110,Y -445.868,Z 1136.571,A 0.000,B 0.000,C 90.000,E1 102.771} C_DIS
LIN {X 0.075,Y -466.133,Z 1136.560,A 0.000,B 0.000,C 90.000,E1 100.782} C_DIS
LIN {X 0.099,Y -468.673,Z 1136.559,A 0.000,B 0.000,C 90.000,E1 100.546} C_DIS
LIN {X 0.122,Y -470.753,Z 1136.557,A 0.000,B 0.000,C 90.000,E1 100.310} C_DIS
LIN {X -0.026,Y -472.453,Z 1136.556,A 0.000,B 0.000,C 90.000,E1 100.074} C_DIS
LIN {X -0.257,Y -473.728,Z 1136.555,A 0.000,B 0.000,C 90.000,E1 99.849} C_DIS
LIN {X -0.068,Y -475.308,Z 1136.552,A 0.000,B 0.000,C 90.000,E1 99.321} C_DIS
LIN {X 0.053,Y -475.833,Z 1136.549,A 0.000,B 0.000,C 90.000,E1 98.803} C_DIS
LIN {X 0.254,Y -475.393,Z 1136.546,A 0.000,B 0.000,C 90.000,E1 98.276} C_DIS
LIN {X -0.083,Y -473.924,Z 1136.543,A 0.000,B 0.000,C 90.000,E1 97.814} C_DIS
LIN {X 0.187,Y -472.728,Z 1136.542,A 0.000,B 0.000,C 90.000,E1 97.530} C_DIS
LIN {X 0.050,Y -471.137,Z 1136.541,A 0.000,B 0.000,C 90.000,E1 97.296} C_DIS
LIN {X 0.155,Y -454.801,Z 1136.528,A 0.000,B 0.000,C 90.000,E1 94.992} C_DIS
LIN {X -0.183,Y -439.113,Z 1136.515,A 0.000,B 0.000,C 90.000,E1 92.694} C_DIS
LIN {X -0.136,Y -419.841,Z 1136.497,A 0.000,B 0.000,C 90.000,E1 89.484} C_DIS
LIN {X -0.188,Y -408.084,Z 1136.485,A 0.000,B 0.000,C 90.000,E1 87.306} C_DIS
LIN {X -0.140,Y -397.576,Z 1136.474,A 0.000,B 0.000,C 90.000,E1 85.355} C_DIS
LIN {X 0.145,Y -385.678,Z 1136.462,A 0.000,B 0.000,C 90.000,E1 83.053} C_DIS
LIN {X -0.164,Y -376.682,Z 1136.452,A 0.000,B 0.000,C 90.000,E1 81.376} C_DIS
LIN {X -0.198,Y -367.430,Z 1136.442,A 0.000,B 0.000,C 90.000,E1 79.634} C_DIS
LIN {X 0.059,Y -359.518,Z 1136.434,A 0.000,B 0.000,C 90.000,E1 78.117} C_DIS
LIN {X -0.127,Y -348.008,Z 1136.422,A 0.000,B 0.000,C 90.000,E1 76.047} C_DIS
LIN {X 0.121,Y -336.514,Z 1136.411,A 0.000,B 0.000,C 90.000,E1 73.866} C_DIS
LIN {X -0.071,Y -323.674,Z 1136.397,A 0.000,B 0.000,C 90.000,E1 71.402} C_DIS
LIN {X 0.099,Y -307.172,Z 1136.377,A 0.000,B 0.000,C 90.000,E1 67.847} C_DIS
LIN {X -0.067,Y -294.485,Z 1136.361,A 0.000,B 0.000,C 90.000,E1 64.921} C_DIS
LIN {X -0.083,Y -282.275,Z 1136.344,A 0.000,B 0.000,C 90.000,E1 61.897} C_DIS
LIN {X -0.022,Y -270.632,Z 1136.327,A 0.000,B 0.000,C 90.000,E1 58.791} C_DIS
LIN {X 0.123,Y -259.499,Z 1136.309,A 0.000,B 0.000,C 90.000,E1 55.595} C_DIS
LIN {X -0.010,Y -247.780,Z 1136.289,A 0.000,B 0.000,C 90.000,E1 52.029} C_DIS
LIN {X -0.012,Y -238.163,Z 1136.271,A 0.000,B 0.000,C 90.000,E1 48.728} C_DIS
LIN {X 0.040,Y -230.207,Z 1136.254,A 0.000,B 0.000,C 90.000,E1 45.729} C_DIS
LIN {X 0.076,Y -220.816,Z 1136.233,A 0.000,B 0.000,C 90.000,E1 41.919} C_DIS
LIN {X -0.120,Y -212.026,Z 1136.211,A 0.000,B 0.000,C 90.000,E1 38.096} C_DIS
LIN {X -0.011,Y -203.824,Z 1136.190,A 0.000,B 0.000,C 90.000,E1 34.119} C_DIS
LIN {X 0.069,Y -196.514,Z 1136.167,A 0.000,B 0.000,C 90.000,E1 30.079} C_DIS
LIN {X 0.060,Y -191.300,Z 1136.149,A 0.000,B 0.000,C 90.000,E1 26.821} C_DIS
LIN {X -0.015,Y -185.707,Z 1136.126,A 0.000,B 0.000,C 90.000,E1 22.717} C_DIS
LIN {X -0.030,Y -181.033,Z 1136.103,A 0.000,B 0.000,C 90.000,E1 18.544} C_DIS
LIN {X 0.040,Y -177.354,Z 1136.079,A 0.000,B 0.000,C 90.000,E1 14.300} C_DIS
LIN {X -0.011,Y -174.375,Z 1136.051,A 0.000,B 0.000,C 90.000,E1 9.208} C_DIS
LIN {X -0.031,Y -172.739,Z 1135.997,A 0.000,B 0.000,C 90.000,E1 359.542} C_DIS
LIN {X 0.056,Y -174.759,Z 1135.959,A 0.000,B 0.000,C 90.000,E1 352.648} C_DIS
LIN {X 0.073,Y -177.942,Z 1135.931,A 0.000,B 0.000,C 90.000,E1 347.521} C_DIS
LIN {X -0.049,Y -181.586,Z 1135.907,A 0.000,B 0.000,C 90.000,E1 343.323} C_DIS
LIN {X 0.083,Y -186.055,Z 1135.884,A 0.000,B 0.000,C 90.000,E1 339.082} C_DIS
LIN {X -0.069,Y -191.460,Z 1135.861,A 0.000,B 0.000,C 90.000,E1 334.973} C_DIS
LIN {X 0.081,Y -196.480,Z 1135.843,A 0.000,B 0.000,C 90.000,E1 331.641} C_DIS
LIN {X 0.024,Y -202.110,Z 1135.824,A 0.000,B 0.000,C 90.000,E1 328.408} C_DIS
LIN {X 0.083,Y -208.345,Z 1135.807,A 0.000,B 0.000,C 90.000,E1 325.182} C_DIS
LIN {X 0.035,Y -215.461,Z 1135.789,A 0.000,B 0.000,C 90.000,E1 322.029} C_DIS
LIN {X -0.037,Y -223.366,Z 1135.772,A 0.000,B 0.000,C 90.000,E1 318.933} C_DIS
LIN {X -0.106,Y -232.266,Z 1135.755,A 0.000,B 0.000,C 90.000,E1 315.891} C_DIS
LIN {X 0.053,Y -242.174,Z 1135.738,A 0.000,B 0.000,C 90.000,E1 312.852} C_DIS
LIN {X -0.023,Y -253.279,Z 1135.722,A 0.000,B 0.000,C 90.000,E1 309.930} C_DIS
LIN {X -0.114,Y -265.786,Z 1135.706,A 0.000,B 0.000,C 90.000,E1 307.076} C_DIS
LIN {X -0.040,Y -281.475,Z 1135.688,A 0.000,B 0.000,C 90.000,E1 303.913} C_DIS
LIN {X -0.123,Y -294.687,Z 1135.675,A 0.000,B 0.000,C 90.000,E1 301.544} C_DIS
LIN {X -0.023,Y -311.293,Z 1135.660,A 0.000,B 0.000,C 90.000,E1 298.871} C_DIS
LIN {X 0.010,Y -331.832,Z 1135.644,A 0.000,B 0.000,C 90.000,E1 295.976} C_DIS
LIN {X 0.051,Y -346.791,Z 1135.634,A 0.000,B 0.000,C 90.000,E1 294.131} C_DIS
LIN {X 0.020,Y -359.869,Z 1135.626,A 0.000,B 0.000,C 90.000,E1 292.695} C_DIS
LIN {X -0.069,Y -378.825,Z 1135.616,A 0.000,B 0.000,C 90.000,E1 290.865} C_DIS
LIN {X -0.227,Y -395.402,Z 1135.608,A 0.000,B 0.000,C 90.000,E1 289.396} C_DIS
LIN {X 0.148,Y -406.177,Z 1135.602,A 0.000,B 0.000,C 90.000,E1 288.362} C_DIS
LIN {X -0.150,Y -416.624,Z 1135.597,A 0.000,B 0.000,C 90.000,E1 287.402} C_DIS
LIN {X -0.092,Y -426.746,Z 1135.591,A 0.000,B 0.000,C 90.000,E1 286.370} C_DIS
LIN {X 0.152,Y -434.057,Z 1135.587,A 0.000,B 0.000,C 90.000,E1 285.552} C_DIS
LIN {X -0.008,Y -441.027,Z 1135.582,A 0.000,B 0.000,C 90.000,E1 284.773} C_DIS
LIN {X -0.232,Y -447.380,Z 1135.578,A 0.000,B 0.000,C 90.000,E1 284.008} C_DIS
LIN {X 0.150,Y -453.038,Z 1135.573,A 0.000,B 0.000,C 90.000,E1 283.175} C_DIS
LIN {X 0.033,Y -457.958,Z 1135.569,A 0.000,B 0.000,C 90.000,E1 282.411} C_DIS
LIN {X -0.134,Y -462.207,Z 1135.565,A 0.000,B 0.000,C 90.000,E1 281.658} C_DIS
LIN {X 0.130,Y -467.066,Z 1135.559,A 0.000,B 0.000,C 90.000,E1 280.602} C_DIS
LIN {X 0.049,Y -470.148,Z 1135.555,A 0.000,B 0.000,C 90.000,E1 279.849} C_DIS
LIN {X 0.214,Y -471.944,Z 1135.552,A 0.000,B 0.000,C 90.000,E1 279.321} C_DIS
LIN {X -0.155,Y -473.479,Z 1135.549,A 0.000,B 0.000,C 90.000,E1 278.859} C_DIS
LIN {X -0.042,Y -474.693,Z 1135.546,A 0.000,B 0.000,C 90.000,E1 278.341} C_DIS
LIN {X 0.146,Y -475.614,Z 1135.543,A 0.000,B 0.000,C 90.000,E1 277.814} C_DIS
LIN {X -0.197,Y -476.210,Z 1135.541,A 0.000,B 0.000,C 90.000,E1 277.352} C_DIS
LIN {X -0.062,Y -476.501,Z 1135.538,A 0.000,B 0.000,C 90.000,E1 276.834} C_DIS
LIN {X 0.078,Y -476.430,Z 1135.535,A 0.000,B 0.000,C 90.000,E1 276.315} C_DIS
LIN {X 0.218,Y -476.006,Z 1135.532,A 0.000,B 0.000,C 90.000,E1 275.796} C_DIS
LIN {X -0.116,Y -475.195,Z 1135.530,A 0.000,B 0.000,C 90.000,E1 275.334} C_DIS
LIN {X -0.020,Y -474.022,Z 1135.527,A 0.000,B 0.000,C 90.000,E1 274.821} C_DIS
LIN {X 0.112,Y -472.403,Z 1135.524,A 0.000,B 0.000,C 90.000,E1 274.302} C_DIS
LIN {X 0.233,Y -470.305,Z 1135.521,A 0.000,B 0.000,C 90.000,E1 273.784} C_DIS
LIN {X 0.040,Y -469.022,Z 1135.520,A 0.000,B 0.000,C 90.000,E1 273.555} C_DIS
LIN {X 0.138,Y -465.872,Z 1135.517,A 0.000,B 0.000,C 90.000,E1 273.037} C_DIS
LIN {X 0.192,Y -461.761,Z 1135.514,A 0.000,B 0.000,C 90.000,E1 272.522} C_DIS
LIN {X -0.014,Y -459.241,Z 1135.513,A 0.000,B 0.000,C 90.000,E1 272.293} C_DIS
LIN {X -0.188,Y -456.430,Z 1135.511,A 0.000,B 0.000,C 90.000,E1 272.064} C_DIS
LIN {X -0.216,Y -450.200,Z 1135.509,A 0.000,B 0.000,C 90.000,E1 271.604} C_DIS
LIN {X -0.143,Y -443.609,Z 1135.507,A 0.000,B 0.000,C 90.000,E1 271.203} C_DIS
LIN {X -0.031,Y -436.714,Z 1135.505,A 0.000,B 0.000,C 90.000,E1 270.859} C_DIS
LIN {X 0.056,Y -429.721,Z 1135.503,A 0.000,B 0.000,C 90.000,E1 270.573} C_DIS
LIN {X 0.040,Y -422.683,Z 1135.502,A 0.000,B 0.000,C 90.000,E1 270.344} C_DIS
LIN {X -0.129,Y -415.275,Z 1135.501,A 0.000,B 0.000,C 90.000,E1 270.172} C_DIS
LIN {X -0.050,Y -407.849,Z 1135.500,A 0.000,B 0.000,C 90.000,E1 270.000} C_DIS
LIN {X -0.171,Y -396.351,Z 1135.499,A 0.000,B 0.000,C 90.000,E1 269.828} C_DIS
LIN {X 0.089,Y -388.424,Z 1135.499,A 0.000,B 0.000,C 90.000,E1 269.714} C_DIS
LIN {X -0.136,Y -381.726,Z 1135.498,A 0.000,B 0.000,C 90.000,E1 269.714} C_DIS
LIN {X -0.091,Y -181.487,Z 1135.498,A 0.000,B 0.000,C 90.000,E1 269.714} C_DIS
LIN {X 0.042,Y -180.906,Z 1135.475,A 0.000,B 0.000,C 90.000,E1 265.412} C_DIS
LIN {X -0.081,Y -180.716,Z 1135.470,A 0.000,B 0.000,C 90.000,E1 264.609} C_DIS
LIN {X 0.017,Y -178.804,Z 1135.442,A 0.000,B 0.000,C 90.000,E1 259.511} C_DIS
LIN {X 0.093,Y -175.848,Z 1135.413,A 0.000,B 0.000,C 90.000,E1 254.393} C_DIS
LIN {X 0.052,Y -172.584,Z 1135.390,A 0.000,B 0.000,C 90.000,E1 250.134} C_DIS
LIN {X 0.069,Y -171.474,Z 1135.380,A 0.000,B 0.000,C 90.000,E1 248.411} C_DIS
LIN {X 0.048,Y -167.704,Z 1135.356,A 0.000,B 0.000,C 90.000,E1 244.101} C_DIS
LIN {X 0.061,Y -166.391,Z 1135.347,A 0.000,B 0.000,C 90.000,E1 242.359} C_DIS
LIN {X 0.052,Y -163.118,Z 1135.327,A 0.000,B 0.000,C 90.000,E1 238.869} C_DIS
LIN {X 0.102,Y -161.067,Z 1135.313,A 0.000,B 0.000,C 90.000,E1 236.215} C_DIS
LIN {X -0.011,Y -157.800,Z 1135.293,A 0.000,B 0.000,C 90.000,E1 232.718} C_DIS
LIN {X -0.072,Y -155.836,Z 1135.278,A 0.000,B 0.000,C 90.000,E1 230.070} C_DIS
LIN {X -0.015,Y -152.086,Z 1135.253,A 0.000,B 0.000,C 90.000,E1 225.567} C_DIS
LIN {X 0.004,Y -150.337,Z 1135.238,A 0.000,B 0.000,C 90.000,E1 222.852} C_DIS
LIN {X 0.024,Y -147.077,Z 1135.213,A 0.000,B 0.000,C 90.000,E1 218.302} C_DIS
LIN {X -0.071,Y -145.650,Z 1135.198,A 0.000,B 0.000,C 90.000,E1 215.598} C_DIS
LIN {X -0.068,Y -143.033,Z 1135.172,A 0.000,B 0.000,C 90.000,E1 211.003} C_DIS
LIN {X 0.059,Y -141.657,Z 1135.152,A 0.000,B 0.000,C 90.000,E1 207.257} C_DIS
LIN {X -0.022,Y -139.447,Z 1135.115,A 0.000,B 0.000,C 90.000,E1 200.791} C_DIS
LIN {X 0.031,Y -139.180,Z 1135.105,A 0.000,B 0.000,C 90.000,E1 198.906} C_DIS
LIN {X 0.059,Y -138.320,Z 1135.053,A 0.000,B 0.000,C 90.000,E1 189.557} C_DIS
LIN {X 0.069,Y -139.465,Z 1135.006,A 0.000,B 0.000,C 90.000,E1 181.146} C_DIS
LIN {X 0.010,Y -141.029,Z 1134.975,A 0.000,B 0.000,C 90.000,E1 175.584} C_DIS
LIN {X -0.036,Y -142.396,Z 1134.960,A 0.000,B 0.000,C 90.000,E1 172.818} C_DIS
LIN {X 0.026,Y -144.628,Z 1134.934,A 0.000,B 0.000,C 90.000,E1 168.173} C_DIS
LIN {X -0.055,Y -147.823,Z 1134.909,A 0.000,B 0.000,C 90.000,E1 163.614} C_DIS
LIN {X 0.031,Y -150.514,Z 1134.889,A 0.000,B 0.000,C 90.000,E1 159.934} C_DIS
LIN {X 0.052,Y -153.976,Z 1134.868,A 0.000,B 0.000,C 90.000,E1 156.305} C_DIS
LIN {X -0.028,Y -157.388,Z 1134.849,A 0.000,B 0.000,C 90.000,E1 152.743} C_DIS
LIN {X -0.085,Y -161.592,Z 1134.829,A 0.000,B 0.000,C 90.000,E1 149.203} C_DIS
LIN {X -0.075,Y -165.789,Z 1134.809,A 0.000,B 0.000,C 90.000,E1 145.674} C_DIS
LIN {X -0.089,Y -170.750,Z 1134.790,A 0.000,B 0.000,C 90.000,E1 142.190} C_DIS
LIN {X 0.069,Y -175.622,Z 1134.771,A 0.000,B 0.000,C 90.000,E1 138.690} C_DIS
LIN {X -0.062,Y -181.238,Z 1134.752,A 0.000,B 0.000,C 90.000,E1 135.324} C_DIS
LIN {X 0.069,Y -186.708,Z 1134.733,A 0.000,B 0.000,C 90.000,E1 131.919} C_DIS
LIN {X 0.020,Y -191.308,Z 1134.719,A 0.000,B 0.000,C 90.000,E1 129.439} C_DIS
LIN {X -0.049,Y -197.137,Z 1134.701,A 0.000,B 0.000,C 90.000,E1 126.171} C_DIS
LIN {X -0.075,Y -201.058,Z 1134.690,A 0.000,B 0.000,C 90.000,E1 124.199} C_DIS
LIN {X -0.157,Y -309.767,Z 1134.690,A 0.000,B 0.000,C 90.000,E1 124.199} C_DIS
LIN {X 0.192,Y -311.074,Z 1134.690,A 0.000,B 0.000,C 90.000,E1 124.119} C_DIS
LIN {X 0.133,Y -316.265,Z 1134.688,A 0.000,B 0.000,C 90.000,E1 123.913} C_DIS
LIN {X 0.071,Y -318.907,Z 1134.687,A 0.000,B 0.000,C 90.000,E1 123.706} C_DIS
LIN {X -0.034,Y -322.695,Z 1134.685,A 0.000,B 0.000,C 90.000,E1 123.245} C_DIS
LIN {X 0.046,Y -324.450,Z 1134.683,A 0.000,B 0.000,C 90.000,E1 122.911} C_DIS
LIN {X -0.050,Y -326.955,Z 1134.679,A 0.000,B 0.000,C 90.000,E1 122.291} C_DIS
LIN {X -0.026,Y -337.823,Z 1134.664,A 0.000,B 0.000,C 90.000,E1 119.461} C_DIS
LIN {X -0.053,Y -350.068,Z 1134.648,A 0.000,B 0.000,C 90.000,E1 116.693} C_DIS
LIN {X 0.122,Y -363.803,Z 1134.633,A 0.000,B 0.000,C 90.000,E1 113.951} C_DIS
LIN {X 0.134,Y -377.355,Z 1134.620,A 0.000,B 0.000,C 90.000,E1 111.589} C_DIS
LIN {X -0.156,Y -392.274,Z 1134.607,A 0.000,B 0.000,C 90.000,E1 109.322} C_DIS
LIN {X 0.036,Y -408.662,Z 1134.595,A 0.000,B 0.000,C 90.000,E1 107.040} C_DIS
LIN {X 0.135,Y -426.638,Z 1134.583,A 0.000,B 0.000,C 90.000,E1 104.828} C_DIS
LIN {X 0.053,Y -446.181,Z 1134.571,A 0.000,B 0.000,C 90.000,E1 102.715} C_DIS
LIN {X -0.163,Y -468.964,Z 1134.558,A 0.000,B 0.000,C 90.000,E1 100.546} C_DIS
LIN {X -0.138,Y -470.957,Z 1134.557,A 0.000,B 0.000,C 90.000,E1 100.310} C_DIS
LIN {X 0.180,Y -472.595,Z 1134.556,A 0.000,B 0.000,C 90.000,E1 100.018} C_DIS
LIN {X -0.050,Y -473.823,Z 1134.554,A 0.000,B 0.000,C 90.000,E1 99.792} C_DIS
LIN {X 0.142,Y -475.327,Z 1134.552,A 0.000,B 0.000,C 90.000,E1 99.265} C_DIS
LIN {X -0.206,Y -475.789,Z 1134.549,A 0.000,B 0.000,C 90.000,E1 98.803} C_DIS
LIN {X -0.005,Y -475.287,Z 1134.546,A 0.000,B 0.000,C 90.000,E1 98.276} C_DIS
LIN {X 0.128,Y -473.745,Z 1134.543,A 0.000,B 0.000,C 90.000,E1 97.757} C_DIS
LIN {X -0.071,Y -472.503,Z 1134.542,A 0.000,B 0.000,C 90.000,E1 97.530} C_DIS
LIN {X 0.113,Y -468.991,Z 1134.539,A 0.000,B 0.000,C 90.000,E1 97.004} C_DIS
LIN {X -0.101,Y -454.544,Z 1134.528,A 0.000,B 0.000,C 90.000,E1 94.992} C_DIS
LIN {X -0.178,Y -440.508,Z 1134.516,A 0.000,B 0.000,C 90.000,E1 92.922} C_DIS
LIN {X -0.086,Y -421.121,Z 1134.498,A 0.000,B 0.000,C 90.000,E1 89.714} C_DIS
LIN {X -0.030,Y -407.811,Z 1134.485,A 0.000,B 0.000,C 90.000,E1 87.249} C_DIS
LIN {X 0.007,Y -397.319,Z 1134.474,A 0.000,B 0.000,C 90.000,E1 85.298} C_DIS
LIN {X -0.102,Y -385.419,Z 1134.461,A 0.000,B 0.000,C 90.000,E1 83.053} C_DIS
LIN {X -0.038,Y -376.398,Z 1134.452,A 0.000,B 0.000,C 90.000,E1 81.319} C_DIS
LIN {X -0.007,Y -368.719,Z 1134.444,A 0.000,B 0.000,C 90.000,E1 79.859} C_DIS
LIN {X -0.158,Y -360.825,Z 1134.435,A 0.000,B 0.000,C 90.000,E1 78.409} C_DIS
LIN {X -0.049,Y -349.339,Z 1134.424,A 0.000,B 0.000,C 90.000,E1 76.297} C_DIS
LIN {X -0.021,Y -337.844,Z 1134.412,A 0.000,B 0.000,C 90.000,E1 74.157} C_DIS
LIN {X 0.138,Y -324.941,Z 1134.398,A 0.000,B 0.000,C 90.000,E1 71.638} C_DIS
LIN {X -0.051,Y -308.313,Z 1134.379,A 0.000,B 0.000,C 90.000,E1 68.156} C_DIS
LIN {X 0.086,Y -295.576,Z 1134.362,A 0.000,B 0.000,C 90.000,E1 65.177} C_DIS
LIN {X 0.124,Y -284.653,Z 1134.347,A 0.000,B 0.000,C 90.000,E1 62.487} C_DIS
LIN {X 0.100,Y -272.873,Z 1134.330,A 0.000,B 0.000,C 90.000,E1 59.410} C_DIS
LIN {X 0.029,Y -262.864,Z 1134.315,A 0.000,B 0.000,C 90.000,E1 56.628} C_DIS
LIN {X 0.001,Y -253.225,Z 1134.299,A 0.000,B 0.000,C 90.000,E1 53.783} C_DIS
LIN {X -0.020,Y -244.134,Z 1134.283,A 0.000,B 0.000,C 90.000,E1 50.884} C_DIS
LIN {X -0.020,Y -233.800,Z 1134.262,A 0.000,B 0.000,C 90.000,E1 47.187} C_DIS
LIN {X -0.078,Y -226.036,Z 1134.245,A 0.000,B 0.000,C 90.000,E1 44.190} C_DIS
LIN {X 0.009,Y -216.873,Z 1134.224,A 0.000,B 0.000,C 90.000,E1 40.334} C_DIS
LIN {X 0.022,Y -208.306,Z 1134.202,A 0.000,B 0.000,C 90.000,E1 36.423} C_DIS
LIN {X 0.023,Y -201.919,Z 1134.185,A 0.000,B 0.000,C 90.000,E1 33.245} C_DIS
LIN {X 0.044,Y -194.763,Z 1134.162,A 0.000,B 0.000,C 90.000,E1 29.205} C_DIS
LIN {X -0.100,Y -189.733,Z 1134.144,A 0.000,B 0.000,C 90.000,E1 25.976} C_DIS
LIN {X -0.017,Y -185.335,Z 1134.126,A 0.000,B 0.000,C 90.000,E1 22.642} C_DIS
LIN {X -0.050,Y -180.678,Z 1134.103,A 0.000,B 0.000,C 90.000,E1 18.471} C_DIS
LIN {X -0.043,Y -177.015,Z 1134.079,A 0.000,B 0.000,C 90.000,E1 14.245} C_DIS
LIN {X 0.069,Y -174.053,Z 1134.051,A 0.000,B 0.000,C 90.000,E1 9.095} C_DIS
LIN {X 0.041,Y -174.429,Z 1133.959,A 0.000,B 0.000,C 90.000,E1 352.648} C_DIS
LIN {X 0.046,Y -177.603,Z 1133.931,A 0.000,B 0.000,C 90.000,E1 347.521} C_DIS
LIN {X -0.087,Y -181.255,Z 1133.907,A 0.000,B 0.000,C 90.000,E1 343.323} C_DIS
LIN {X 0.033,Y -185.680,Z 1133.884,A 0.000,B 0.000,C 90.000,E1 339.082} C_DIS
LIN {X 0.040,Y -191.105,Z 1133.861,A 0.000,B 0.000,C 90.000,E1 334.921} C_DIS
LIN {X 0.008,Y -196.157,Z 1133.842,A 0.000,B 0.000,C 90.000,E1 331.641} C_DIS
LIN {X -0.060,Y -201.814,Z 1133.824,A 0.000,B 0.000,C 90.000,E1 328.408} C_DIS
LIN {X -0.010,Y -208.076,Z 1133.807,A 0.000,B 0.000,C 90.000,E1 325.182} C_DIS
LIN {X 0.101,Y -215.216,Z 1133.789,A 0.000,B 0.000,C 90.000,E1 321.984} C_DIS
LIN {X -0.003,Y -223.146,Z 1133.772,A 0.000,B 0.000,C 90.000,E1 318.895} C_DIS
LIN {X 0.099,Y -232.082,Z 1133.755,A 0.000,B 0.000,C 90.000,E1 315.810} C_DIS
LIN {X -0.081,Y -242.001,Z 1133.738,A 0.000,B 0.000,C 90.000,E1 312.852} C_DIS
LIN {X 0.016,Y -251.695,Z 1133.724,A 0.000,B 0.000,C 90.000,E1 310.253} C_DIS
LIN {X 0.054,Y -264.105,Z 1133.708,A 0.000,B 0.000,C 90.000,E1 307.363} C_DIS
LIN {X 0.082,Y -279.691,Z 1133.690,A 0.000,B 0.000,C 90.000,E1 304.199} C_DIS
LIN {X 0.110,Y -294.735,Z 1133.675,A 0.000,B 0.000,C 90.000,E1 301.465} C_DIS
LIN {X 0.070,Y -311.409,Z 1133.660,A 0.000,B 0.000,C 90.000,E1 298.821} C_DIS
LIN {X -0.178,Y -331.978,Z 1133.644,A 0.000,B 0.000,C 90.000,E1 295.976} C_DIS
LIN {X 0.185,Y -346.920,Z 1133.634,A 0.000,B 0.000,C 90.000,E1 294.079} C_DIS
LIN {X -0.169,Y -362.313,Z 1133.625,A 0.000,B 0.000,C 90.000,E1 292.461} C_DIS
LIN {X 0.042,Y -389.341,Z 1133.610,A 0.000,B 0.000,C 90.000,E1 289.885} C_DIS
LIN {X 0.004,Y -402.952,Z 1133.604,A 0.000,B 0.000,C 90.000,E1 288.671} C_DIS
LIN {X -0.063,Y -413.462,Z 1133.598,A 0.000,B 0.000,C 90.000,E1 287.692} C_DIS
LIN {X 0.133,Y -421.096,Z 1133.594,A 0.000,B 0.000,C 90.000,E1 286.913} C_DIS
LIN {X 0.066,Y -428.622,Z 1133.590,A 0.000,B 0.000,C 90.000,E1 286.150} C_DIS
LIN {X 0.146,Y -438.266,Z 1133.584,A 0.000,B 0.000,C 90.000,E1 285.079} C_DIS
LIN {X 0.020,Y -444.895,Z 1133.579,A 0.000,B 0.000,C 90.000,E1 284.300} C_DIS
LIN {X -0.169,Y -450.896,Z 1133.575,A 0.000,B 0.000,C 90.000,E1 283.536} C_DIS
LIN {X 0.146,Y -456.118,Z 1133.571,A 0.000,B 0.000,C 90.000,E1 282.715} C_DIS
LIN {X 0.059,Y -460.707,Z 1133.566,A 0.000,B 0.000,C 90.000,E1 281.951} C_DIS
LIN {X 0.014,Y -464.627,Z 1133.562,A 0.000,B 0.000,C 90.000,E1 281.186} C_DIS
LIN {X -0.006,Y -468.085,Z 1133.558,A 0.000,B 0.000,C 90.000,E1 280.423} C_DIS
LIN {X 0.068,Y -470.123,Z 1133.555,A 0.000,B 0.000,C 90.000,E1 279.905} C_DIS
LIN {X 0.232,Y -471.974,Z 1133.552,A 0.000,B 0.000,C 90.000,E1 279.378} C_DIS
LIN {X -0.137,Y -473.528,Z 1133.549,A 0.000,B 0.000,C 90.000,E1 278.916} C_DIS
LIN {X -0.026,Y -474.788,Z 1133.547,A 0.000,B 0.000,C 90.000,E1 278.398} C_DIS
LIN {X 0.163,Y -475.744,Z 1133.544,A 0.000,B 0.000,C 90.000,E1 277.871} C_DIS
LIN {X -0.180,Y -476.381,Z 1133.541,A 0.000,B 0.000,C 90.000,E1 277.409} C_DIS
LIN {X -0.044,Y -476.704,Z 1133.538,A 0.000,B 0.000,C 90.000,E1 276.891} C_DIS
LIN {X 0.096,Y -476.679,Z 1133.536,A 0.000,B 0.000,C 90.000,E1 276.372} C_DIS
LIN {X 0.237,Y -476.313,Z 1133.533,A 0.000,B 0.000,C 90.000,E1 275.853} C_DIS
LIN {X -0.097,Y -475.598,Z 1133.530,A 0.000,B 0.000,C 90.000,E1 275.391} C_DIS
LIN {X 0.001,Y -474.506,Z 1133.527,A 0.000,B 0.000,C 90.000,E1 274.878} C_DIS
LIN {X 0.135,Y -472.982,Z 1133.524,A 0.000,B 0.000,C 90.000,E1 274.359} C_DIS
LIN {X -0.211,Y -470.999,Z 1133.521,A 0.000,B 0.000,C 90.000,E1 273.898} C_DIS
LIN {X -0.125,Y -468.349,Z 1133.519,A 0.000,B 0.000,C 90.000,E1 273.383} C_DIS
LIN {X 0.168,Y -466.766,Z 1133.517,A 0.000,B 0.000,C 90.000,E1 273.094} C_DIS
LIN {X 0.226,Y -462.829,Z 1133.515,A 0.000,B 0.000,C 90.000,E1 272.579} C_DIS
LIN {X 0.021,Y -460.457,Z 1133.513,A 0.000,B 0.000,C 90.000,E1 272.350} C_DIS
LIN {X -0.192,Y -457.723,Z 1133.512,A 0.000,B 0.000,C 90.000,E1 272.121} C_DIS
LIN {X 0.053,Y -454.590,Z 1133.510,A 0.000,B 0.000,C 90.000,E1 271.835} C_DIS
LIN {X 0.225,Y -448.171,Z 1133.508,A 0.000,B 0.000,C 90.000,E1 271.375} C_DIS
LIN {X 0.019,Y -441.437,Z 1133.506,A 0.000,B 0.000,C 90.000,E1 271.031} C_DIS
LIN {X -0.173,Y -434.363,Z 1133.504,A 0.000,B 0.000,C 90.000,E1 270.745} C_DIS
LIN {X 0.055,Y -427.420,Z 1133.503,A 0.000,B 0.000,C 90.000,E1 270.458} C_DIS
LIN {X 0.117,Y -420.153,Z 1133.501,A 0.000,B 0.000,C 90.000,E1 270.229} C_DIS
LIN {X -0.032,Y -409.437,Z 1133.500,A 0.000,B 0.000,C 90.000,E1 270.000} C_DIS
LIN {X 0.198,Y -397.609,Z 1133.499,A 0.000,B 0.000,C 90.000,E1 269.771} C_DIS
LIN {X -0.097,Y -386.992,Z 1133.498,A 0.000,B 0.000,C 90.000,E1 269.714} C_DIS
LIN {X 0.112,Y -381.224,Z 1133.498,A 0.000,B 0.000,C 90.000,E1 269.656} C_DIS
LIN {X 0.026,Y -181.481,Z 1133.498,A 0.000,B 0.000,C 90.000,E1 269.656} C_DIS
LIN {X 0.019,Y -180.906,Z 1133.474,A 0.000,B 0.000,C 90.000,E1 265.412} C_DIS
LIN {X 0.075,Y -180.713,Z 1133.470,A 0.000,B 0.000,C 90.000,E1 264.552} C_DIS
LIN {X -0.006,Y -178.800,Z 1133.442,A 0.000,B 0.000,C 90.000,E1 259.511} C_DIS
LIN {X 0.070,Y -175.845,Z 1133.413,A 0.000,B 0.000,C 90.000,E1 254.393} C_DIS
LIN {X 0.070,Y -172.036,Z 1133.385,A 0.000,B 0.000,C 90.000,E1 249.263} C_DIS
LIN {X 0.046,Y -171.468,Z 1133.380,A 0.000,B 0.000,C 90.000,E1 248.411} C_DIS
LIN {X 0.026,Y -167.698,Z 1133.356,A 0.000,B 0.000,C 90.000,E1 244.101} C_DIS
LIN {X 0.039,Y -166.383,Z 1133.347,A 0.000,B 0.000,C 90.000,E1 242.359} C_DIS
LIN {X 0.031,Y -163.112,Z 1133.327,A 0.000,B 0.000,C 90.000,E1 238.869} C_DIS
LIN {X 0.081,Y -161.060,Z 1133.313,A 0.000,B 0.000,C 90.000,E1 236.215} C_DIS
LIN {X -0.032,Y -157.795,Z 1133.293,A 0.000,B 0.000,C 90.000,E1 232.718} C_DIS
LIN {X 0.007,Y -155.830,Z 1133.278,A 0.000,B 0.000,C 90.000,E1 230.033} C_DIS
LIN {X -0.036,Y -152.081,Z 1133.253,A 0.000,B 0.000,C 90.000,E1 225.567} C_DIS
LIN {X -0.017,Y -150.332,Z 1133.238,A 0.000,B 0.000,C 90.000,E1 222.852} C_DIS
LIN {X 0.004,Y -147.071,Z 1133.213,A 0.000,B 0.000,C 90.000,E1 218.302} C_DIS
LIN {X -0.091,Y -145.647,Z 1133.198,A 0.000,B 0.000,C 90.000,E1 215.598} C_DIS
LIN {X -0.088,Y -143.029,Z 1133.172,A 0.000,B 0.000,C 90.000,E1 211.003} C_DIS
LIN {X 0.040,Y -141.654,Z 1133.151,A 0.000,B 0.000,C 90.000,E1 207.257} C_DIS
LIN {X -0.041,Y -139.445,Z 1133.115,A 0.000,B 0.000,C 90.000,E1 200.791} C_DIS
LIN {X 0.011,Y -139.178,Z 1133.105,A 0.000,B 0.000,C 90.000,E1 198.906} C_DIS
LIN {X 0.040,Y -138.319,Z 1133.053,A 0.000,B 0.000,C 90.000,E1 189.557} C_DIS
LIN {X 0.049,Y -139.467,Z 1133.006,A 0.000,B 0.000,C 90.000,E1 181.146} C_DIS
LIN {X -0.010,Y -141.033,Z 1132.975,A 0.000,B 0.000,C 90.000,E1 175.584} C_DIS
LIN {X -0.056,Y -142.399,Z 1132.960,A 0.000,B 0.000,C 90.000,E1 172.818} C_DIS
LIN {X 0.006,Y -144.632,Z 1132.934,A 0.000,B 0.000,C 90.000,E1 168.173} C_DIS
LIN {X 0.067,Y -147.828,Z 1132.909,A 0.000,B 0.000,C 90.000,E1 163.559} C_DIS
LIN {X 0.011,Y -150.520,Z 1132.889,A 0.000,B 0.000,C 90.000,E1 159.934} C_DIS
LIN {X 0.031,Y -153.983,Z 1132.868,A 0.000,B 0.000,C 90.000,E1 156.305} C_DIS
LIN {X -0.048,Y -157.396,Z 1132.849,A 0.000,B 0.000,C 90.000,E1 152.743} C_DIS
LIN {X 0.032,Y -161.601,Z 1132.829,A 0.000,B 0.000,C 90.000,E1 149.154} C_DIS
LIN {X -0.096,Y -165.798,Z 1132.809,A 0.000,B 0.000,C 90.000,E1 145.674} C_DIS
LIN {X 0.023,Y -170.762,Z 1132.790,A 0.000,B 0.000,C 90.000,E1 142.145} C_DIS
LIN {X 0.046,Y -175.634,Z 1132.771,A 0.000,B 0.000,C 90.000,E1 138.690} C_DIS
LIN {X -0.084,Y -181.249,Z 1132.752,A 0.000,B 0.000,C 90.000,E1 135.324} C_DIS
LIN {X 0.046,Y -186.720,Z 1132.733,A 0.000,B 0.000,C 90.000,E1 131.919} C_DIS
LIN {X -0.003,Y -191.319,Z 1132.719,A 0.000,B 0.000,C 90.000,E1 129.439} C_DIS
LIN {X -0.073,Y -197.150,Z 1132.701,A 0.000,B 0.000,C 90.000,E1 126.171} C_DIS
LIN {X 0.051,Y -200.997,Z 1132.690,A 0.000,B 0.000,C 90.000,E1 124.199} C_DIS
LIN {X 0.031,Y -309.876,Z 1132.690,A 0.000,B 0.000,C 90.000,E1 124.199} C_DIS
LIN {X 0.053,Y -314.254,Z 1132.689,A 0.000,B 0.000,C 90.000,E1 124.072} C_DIS
LIN {X -0.187,Y -316.334,Z 1132.689,A 0.000,B 0.000,C 90.000,E1 123.992} C_DIS
LIN {X 0.032,Y -319.184,Z 1132.687,A 0.000,B 0.000,C 90.000,E1 123.706} C_DIS
LIN {X -0.002,Y -322.916,Z 1132.685,A 0.000,B 0.000,C 90.000,E1 123.214} C_DIS
LIN {X 0.077,Y -324.588,Z 1132.683,A 0.000,B 0.000,C 90.000,E1 122.880} C_DIS
LIN {X -0.020,Y -327.025,Z 1132.679,A 0.000,B 0.000,C 90.000,E1 122.260} C_DIS
LIN {X 0.122,Y -337.904,Z 1132.663,A 0.000,B 0.000,C 90.000,E1 119.411} C_DIS
LIN {X -0.046,Y -350.162,Z 1132.648,A 0.000,B 0.000,C 90.000,E1 116.668} C_DIS
LIN {X -0.032,Y -363.910,Z 1132.633,A 0.000,B 0.000,C 90.000,E1 113.951} C_DIS
LIN {X -0.022,Y -377.475,Z 1132.620,A 0.000,B 0.000,C 90.000,E1 111.589} C_DIS
LIN {X 0.055,Y -392.408,Z 1132.607,A 0.000,B 0.000,C 90.000,E1 109.268} C_DIS
LIN {X -0.126,Y -408.812,Z 1132.595,A 0.000,B 0.000,C 90.000,E1 107.040} C_DIS
LIN {X -0.031,Y -426.804,Z 1132.582,A 0.000,B 0.000,C 90.000,E1 104.828} C_DIS
LIN {X -0.013,Y -446.359,Z 1132.571,A 0.000,B 0.000,C 90.000,E1 102.703} C_DIS
LIN {X 0.140,Y -469.121,Z 1132.558,A 0.000,B 0.000,C 90.000,E1 100.489} C_DIS
LIN {X 0.169,Y -471.063,Z 1132.557,A 0.000,B 0.000,C 90.000,E1 100.254} C_DIS
LIN {X 0.023,Y -472.662,Z 1132.556,A 0.000,B 0.000,C 90.000,E1 100.018} C_DIS
LIN {X -0.126,Y -473.861,Z 1132.554,A 0.000,B 0.000,C 90.000,E1 99.782} C_DIS
LIN {X -0.015,Y -475.321,Z 1132.552,A 0.000,B 0.000,C 90.000,E1 99.265} C_DIS
LIN {X 0.107,Y -475.744,Z 1132.549,A 0.000,B 0.000,C 90.000,E1 98.746} C_DIS
LIN {X -0.162,Y -475.202,Z 1132.546,A 0.000,B 0.000,C 90.000,E1 98.276} C_DIS
LIN {X -0.029,Y -473.615,Z 1132.543,A 0.000,B 0.000,C 90.000,E1 97.757} C_DIS
LIN {X -0.227,Y -472.344,Z 1132.542,A 0.000,B 0.000,C 90.000,E1 97.530} C_DIS
LIN {X 0.217,Y -466.959,Z 1132.537,A 0.000,B 0.000,C 90.000,E1 96.720} C_DIS
LIN {X 0.196,Y -454.369,Z 1132.528,A 0.000,B 0.000,C 90.000,E1 94.935} C_DIS
LIN {X 0.107,Y -440.322,Z 1132.516,A 0.000,B 0.000,C 90.000,E1 92.865} C_DIS
LIN {X 0.180,Y -420.948,Z 1132.498,A 0.000,B 0.000,C 90.000,E1 89.656} C_DIS
LIN {X -0.185,Y -407.618,Z 1132.485,A 0.000,B 0.000,C 90.000,E1 87.249} C_DIS
LIN {X -0.147,Y -397.138,Z 1132.474,A 0.000,B 0.000,C 90.000,E1 85.298} C_DIS
LIN {X 0.126,Y -385.232,Z 1132.461,A 0.000,B 0.000,C 90.000,E1 82.996} C_DIS
LIN {X -0.135,Y -376.192,Z 1132.452,A 0.000,B 0.000,C 90.000,E1 81.310} C_DIS
LIN {X -0.160,Y -368.524,Z 1132.443,A 0.000,B 0.000,C 90.000,E1 79.859} C_DIS
LIN {X 0.086,Y -358.963,Z 1132.434,A 0.000,B 0.000,C 90.000,E1 78.049} C_DIS
LIN {X -0.118,Y -349.114,Z 1132.424,A 0.000,B 0.000,C 90.000,E1 76.284} C_DIS
LIN {X -0.174,Y -337.608,Z 1132.412,A 0.000,B 0.000,C 90.000,E1 74.157} C_DIS
LIN {X -0.015,Y -324.696,Z 1132.398,A 0.000,B 0.000,C 90.000,E1 71.638} C_DIS
LIN {X -0.122,Y -309.542,Z 1132.380,A 0.000,B 0.000,C 90.000,E1 68.465} C_DIS
LIN {X 0.058,Y -296.763,Z 1132.364,A 0.000,B 0.000,C 90.000,E1 65.485} C_DIS
LIN {X -0.028,Y -284.443,Z 1132.347,A 0.000,B 0.000,C 90.000,E1 62.487} C_DIS
LIN {X -0.051,Y -272.646,Z 1132.330,A 0.000,B 0.000,C 90.000,E1 59.410} C_DIS
LIN {X -0.123,Y -262.623,Z 1132.314,A 0.000,B 0.000,C 90.000,E1 56.628} C_DIS
LIN {X -0.001,Y -252.970,Z 1132.299,A 0.000,B 0.000,C 90.000,E1 53.749} C_DIS
LIN {X -0.019,Y -243.847,Z 1132.282,A 0.000,B 0.000,C 90.000,E1 50.848} C_DIS
LIN {X -0.016,Y -233.523,Z 1132.262,A 0.000,B 0.000,C 90.000,E1 47.148} C_DIS
LIN {X -0.041,Y -223.839,Z 1132.241,A 0.000,B 0.000,C 90.000,E1 43.380} C_DIS
LIN {X -0.010,Y -216.560,Z 1132.224,A 0.000,B 0.000,C 90.000,E1 40.297} C_DIS
LIN {X 0.026,Y -207.963,Z 1132.202,A 0.000,B 0.000,C 90.000,E1 36.377} C_DIS
LIN {X -0.033,Y -201.581,Z 1132.184,A 0.000,B 0.000,C 90.000,E1 33.214} C_DIS
LIN {X 0.044,Y -194.413,Z 1132.162,A 0.000,B 0.000,C 90.000,E1 29.155} C_DIS
LIN {X -0.020,Y -189.381,Z 1132.144,A 0.000,B 0.000,C 90.000,E1 25.899} C_DIS
LIN {X -0.025,Y -184.983,Z 1132.125,A 0.000,B 0.000,C 90.000,E1 22.589} C_DIS
LIN {X -0.064,Y -180.338,Z 1132.102,A 0.000,B 0.000,C 90.000,E1 18.417} C_DIS
LIN {X -0.020,Y -176.701,Z 1132.079,A 0.000,B 0.000,C 90.000,E1 14.175} C_DIS
LIN {X 0.068,Y -173.750,Z 1132.050,A 0.000,B 0.000,C 90.000,E1 9.029} C_DIS
LIN {X 0.056,Y -174.544,Z 1131.954,A 0.000,B 0.000,C 90.000,E1 351.781} C_DIS
LIN {X -0.076,Y -177.917,Z 1131.926,A 0.000,B 0.000,C 90.000,E1 346.700} C_DIS
LIN {X 0.069,Y -181.752,Z 1131.902,A 0.000,B 0.000,C 90.000,E1 342.417} C_DIS
LIN {X 0.033,Y -186.332,Z 1131.879,A 0.000,B 0.000,C 90.000,E1 338.230} C_DIS
LIN {X 0.041,Y -191.965,Z 1131.856,A 0.000,B 0.000,C 90.000,E1 334.076} C_DIS
LIN {X 0.032,Y -197.215,Z 1131.838,A 0.000,B 0.000,C 90.000,E1 330.795} C_DIS
LIN {X -0.001,Y -204.532,Z 1131.815,A 0.000,B 0.000,C 90.000,E1 326.755} C_DIS
LIN {X -0.053,Y -211.284,Z 1131.798,A 0.000,B 0.000,C 90.000,E1 323.577} C_DIS
LIN {X -0.019,Y -219.837,Z 1131.778,A 0.000,B 0.000,C 90.000,E1 320.033} C_DIS
LIN {X 0.007,Y -228.403,Z 1131.761,A 0.000,B 0.000,C 90.000,E1 316.944} C_DIS
LIN {X -0.107,Y -237.962,Z 1131.744,A 0.000,B 0.000,C 90.000,E1 313.947} C_DIS
LIN {X 0.054,Y -248.657,Z 1131.728,A 0.000,B 0.000,C 90.000,E1 310.943} C_DIS
LIN {X 0.142,Y -259.206,Z 1131.713,A 0.000,B 0.000,C 90.000,E1 308.382} C_DIS
LIN {X -0.111,Y -272.585,Z 1131.698,A 0.000,B 0.000,C 90.000,E1 305.598} C_DIS
LIN {X 0.009,Y -288.958,Z 1131.680,A 0.000,B 0.000,C 90.000,E1 302.467} C_DIS
LIN {X -0.065,Y -300.906,Z 1131.669,A 0.000,B 0.000,C 90.000,E1 300.463} C_DIS
LIN {X -0.048,Y -320.452,Z 1131.653,A 0.000,B 0.000,C 90.000,E1 297.513} C_DIS
LIN {X 0.036,Y -334.579,Z 1131.642,A 0.000,B 0.000,C 90.000,E1 295.591} C_DIS
LIN {X -0.013,Y -347.086,Z 1131.634,A 0.000,B 0.000,C 90.000,E1 294.079} C_DIS
LIN {X -0.143,Y -360.393,Z 1131.626,A 0.000,B 0.000,C 90.000,E1 292.642} C_DIS
LIN {X -0.110,Y -387.637,Z 1131.611,A 0.000,B 0.000,C 90.000,E1 290.047} C_DIS
LIN {X 0.196,Y -401.338,Z 1131.604,A 0.000,B 0.000,C 90.000,E1 288.779} C_DIS
LIN {X 0.024,Y -411.936,Z 1131.599,A 0.000,B 0.000,C 90.000,E1 287.819} C_DIS
LIN {X 0.080,Y -422.234,Z 1131.593,A 0.000,B 0.000,C 90.000,E1 286.804} C_DIS
LIN {X 0.099,Y -429.746,Z 1131.589,A 0.000,B 0.000,C 90.000,E1 286.024} C_DIS
LIN {X -0.033,Y -436.993,Z 1131.585,A 0.000,B 0.000,C 90.000,E1 285.245} C_DIS
LIN {X 0.136,Y -443.806,Z 1131.580,A 0.000,B 0.000,C 90.000,E1 284.426} C_DIS
LIN {X 0.054,Y -449.945,Z 1131.576,A 0.000,B 0.000,C 90.000,E1 283.647} C_DIS
LIN {X -0.092,Y -455.373,Z 1131.572,A 0.000,B 0.000,C 90.000,E1 282.883} C_DIS
LIN {X -0.185,Y -460.103,Z 1131.567,A 0.000,B 0.000,C 90.000,E1 282.119} C_DIS
LIN {X 0.209,Y -464.170,Z 1131.563,A 0.000,B 0.000,C 90.000,E1 281.299} C_DIS
LIN {X 0.103,Y -467.707,Z 1131.559,A 0.000,B 0.000,C 90.000,E1 280.546} C_DIS
LIN {X 0.029,Y -470.805,Z 1131.554,A 0.000,B 0.000,C 90.000,E1 279.792} C_DIS
LIN {X 0.197,Y -472.580,Z 1131.552,A 0.000,B 0.000,C 90.000,E1 279.265} C_DIS
LIN {X -0.168,Y -474.067,Z 1131.549,A 0.000,B 0.000,C 90.000,E1 278.803} C_DIS
LIN {X 0.018,Y -475.242,Z 1131.546,A 0.000,B 0.000,C 90.000,E1 278.276} C_DIS
LIN {X 0.142,Y -476.121,Z 1131.543,A 0.000,B 0.000,C 90.000,E1 277.757} C_DIS
LIN {X -0.198,Y -476.701,Z 1131.540,A 0.000,B 0.000,C 90.000,E1 277.296} C_DIS
LIN {X -0.058,Y -476.942,Z 1131.538,A 0.000,B 0.000,C 90.000,E1 276.777} C_DIS
LIN {X 0.084,Y -476.865,Z 1131.535,A 0.000,B 0.000,C 90.000,E1 276.258} C_DIS
LIN {X 0.227,Y -476.455,Z 1131.532,A 0.000,B 0.000,C 90.000,E1 275.739} C_DIS
LIN {X -0.104,Y -475.679,Z 1131.529,A 0.000,B 0.000,C 90.000,E1 275.277} C_DIS
LIN {X 0.035,Y -474.509,Z 1131.526,A 0.000,B 0.000,C 90.000,E1 274.759} C_DIS
LIN {X 0.130,Y -472.941,Z 1131.524,A 0.000,B 0.000,C 90.000,E1 274.245} C_DIS
LIN {X -0.216,Y -470.873,Z 1131.521,A 0.000,B 0.000,C 90.000,E1 273.784} C_DIS
LIN {X -0.129,Y -468.094,Z 1131.518,A 0.000,B 0.000,C 90.000,E1 273.269} C_DIS
LIN {X -0.035,Y -464.536,Z 1131.515,A 0.000,B 0.000,C 90.000,E1 272.751} C_DIS
LIN {X 0.015,Y -459.806,Z 1131.512,A 0.000,B 0.000,C 90.000,E1 272.236} C_DIS
LIN {X -0.164,Y -456.982,Z 1131.511,A 0.000,B 0.000,C 90.000,E1 272.007} C_DIS
LIN {X -0.184,Y -450.771,Z 1131.508,A 0.000,B 0.000,C 90.000,E1 271.547} C_DIS
LIN {X -0.077,Y -444.171,Z 1131.506,A 0.000,B 0.000,C 90.000,E1 271.146} C_DIS
LIN {X 0.058,Y -437.297,Z 1131.505,A 0.000,B 0.000,C 90.000,E1 270.802} C_DIS
LIN {X 0.135,Y -430.264,Z 1131.503,A 0.000,B 0.000,C 90.000,E1 270.516} C_DIS
LIN {X 0.078,Y -423.248,Z 1131.502,A 0.000,B 0.000,C 90.000,E1 270.286} C_DIS
LIN {X -0.092,Y -415.697,Z 1131.501,A 0.000,B 0.000,C 90.000,E1 270.115} C_DIS
LIN {X 0.023,Y -408.316,Z 1131.500,A 0.000,B 0.000,C 90.000,E1 269.943} C_DIS
LIN {X -0.077,Y -400.795,Z 1131.499,A 0.000,B 0.000,C 90.000,E1 269.828} C_DIS
LIN {X -0.161,Y -389.018,Z 1131.498,A 0.000,B 0.000,C 90.000,E1 269.714} C_DIS
LIN {X 0.021,Y -382.294,Z 1131.498,A 0.000,B 0.000,C 90.000,E1 269.656} C_DIS
LIN {X -0.013,Y -181.478,Z 1131.498,A 0.000,B 0.000,C 90.000,E1 269.656} C_DIS
LIN {X -0.049,Y -180.906,Z 1131.474,A 0.000,B 0.000,C 90.000,E1 265.412} C_DIS
LIN {X 0.025,Y -180.703,Z 1131.470,A 0.000,B 0.000,C 90.000,E1 264.546} C_DIS
LIN {X -0.073,Y -178.788,Z 1131.442,A 0.000,B 0.000,C 90.000,E1 259.511} C_DIS
LIN {X 0.004,Y -175.834,Z 1131.413,A 0.000,B 0.000,C 90.000,E1 254.393} C_DIS
LIN {X 0.004,Y -172.023,Z 1131.385,A 0.000,B 0.000,C 90.000,E1 249.263} C_DIS
LIN {X -0.020,Y -171.448,Z 1131.380,A 0.000,B 0.000,C 90.000,E1 248.411} C_DIS
LIN {X 0.035,Y -167.682,Z 1131.356,A 0.000,B 0.000,C 90.000,E1 244.076} C_DIS
LIN {X -0.025,Y -166.360,Z 1131.346,A 0.000,B 0.000,C 90.000,E1 242.359} C_DIS
LIN {X -0.033,Y -163.093,Z 1131.327,A 0.000,B 0.000,C 90.000,E1 238.869} C_DIS
LIN {X 0.018,Y -161.037,Z 1131.312,A 0.000,B 0.000,C 90.000,E1 236.215} C_DIS
LIN {X 0.002,Y -157.776,Z 1131.293,A 0.000,B 0.000,C 90.000,E1 232.683} C_DIS
LIN {X 0.065,Y -155.813,Z 1131.278,A 0.000,B 0.000,C 90.000,E1 229.989} C_DIS
LIN {X 0.012,Y -152.065,Z 1131.253,A 0.000,B 0.000,C 90.000,E1 225.526} C_DIS
LIN {X -0.077,Y -150.314,Z 1131.238,A 0.000,B 0.000,C 90.000,E1 222.852} C_DIS
LIN {X -0.055,Y -147.057,Z 1131.213,A 0.000,B 0.000,C 90.000,E1 218.302} C_DIS
LIN {X 0.053,Y -145.635,Z 1131.197,A 0.000,B 0.000,C 90.000,E1 215.518} C_DIS
LIN {X 0.050,Y -143.017,Z 1131.172,A 0.000,B 0.000,C 90.000,E1 210.924} C_DIS
LIN {X -0.018,Y -141.644,Z 1131.151,A 0.000,B 0.000,C 90.000,E1 207.257} C_DIS
LIN {X 0.032,Y -139.441,Z 1131.115,A 0.000,B 0.000,C 90.000,E1 200.737} C_DIS
LIN {X -0.046,Y -139.173,Z 1131.105,A 0.000,B 0.000,C 90.000,E1 198.906} C_DIS
LIN {X -0.018,Y -138.319,Z 1131.053,A 0.000,B 0.000,C 90.000,E1 189.557} C_DIS
LIN {X -0.009,Y -139.471,Z 1131.006,A 0.000,B 0.000,C 90.000,E1 181.146} C_DIS
LIN {X -0.069,Y -141.043,Z 1130.975,A 0.000,B 0.000,C 90.000,E1 175.584} C_DIS
LIN {X 0.027,Y -142.412,Z 1130.960,A 0.000,B 0.000,C 90.000,E1 172.761} C_DIS
LIN {X -0.053,Y -144.646,Z 1130.934,A 0.000,B 0.000,C 90.000,E1 168.173} C_DIS
LIN {X 0.006,Y -147.842,Z 1130.909,A 0.000,B 0.000,C 90.000,E1 163.559} C_DIS
LIN {X -0.049,Y -150.540,Z 1130.888,A 0.000,B 0.000,C 90.000,E1 159.934} C_DIS
LIN {X -0.031,Y -154.005,Z 1130.868,A 0.000,B 0.000,C 90.000,E1 156.305} C_DIS
LIN {X 0.029,Y -157.420,Z 1130.848,A 0.000,B 0.000,C 90.000,E1 152.692} C_DIS
LIN {X 0.052,Y -161.631,Z 1130.829,A 0.000,B 0.000,C 90.000,E1 149.125} C_DIS
LIN {X 0.070,Y -165.827,Z 1130.809,A 0.000,B 0.000,C 90.000,E1 145.595} C_DIS
LIN {X 0.062,Y -170.796,Z 1130.790,A 0.000,B 0.000,C 90.000,E1 142.110} C_DIS
LIN {X -0.020,Y -175.667,Z 1130.771,A 0.000,B 0.000,C 90.000,E1 138.690} C_DIS
LIN {X -0.024,Y -181.281,Z 1130.752,A 0.000,B 0.000,C 90.000,E1 135.283} C_DIS
LIN {X -0.024,Y -186.759,Z 1130.733,A 0.000,B 0.000,C 90.000,E1 131.919} C_DIS
LIN {X 0.047,Y -191.353,Z 1130.719,A 0.000,B 0.000,C 90.000,E1 129.402} C_DIS
LIN {X -0.027,Y -197.190,Z 1130.701,A 0.000,B 0.000,C 90.000,E1 126.137} C_DIS
LIN {X -0.003,Y -200.942,Z 1130.690,A 0.000,B 0.000,C 90.000,E1 124.246} C_DIS
LIN {X -0.039,Y -309.678,Z 1130.690,A 0.000,B 0.000,C 90.000,E1 124.246} C_DIS
LIN {X -0.078,Y -312.419,Z 1130.690,A 0.000,B 0.000,C 90.000,E1 124.199} C_DIS
LIN {X 0.140,Y -316.936,Z 1130.689,A 0.000,B 0.000,C 90.000,E1 123.913} C_DIS
LIN {X -0.082,Y -319.559,Z 1130.687,A 0.000,B 0.000,C 90.000,E1 123.706} C_DIS
LIN {X -0.043,Y -323.289,Z 1130.684,A 0.000,B 0.000,C 90.000,E1 123.166} C_DIS
LIN {X 0.039,Y -324.844,Z 1130.682,A 0.000,B 0.000,C 90.000,E1 122.832} C_DIS
LIN {X -0.196,Y -338.104,Z 1130.663,A 0.000,B 0.000,C 90.000,E1 119.411} C_DIS
LIN {X -0.054,Y -350.388,Z 1130.648,A 0.000,B 0.000,C 90.000,E1 116.616} C_DIS
LIN {X -0.027,Y -364.166,Z 1130.633,A 0.000,B 0.000,C 90.000,E1 113.898} C_DIS
LIN {X -0.005,Y -377.760,Z 1130.620,A 0.000,B 0.000,C 90.000,E1 111.535} C_DIS
LIN {X 0.086,Y -392.722,Z 1130.607,A 0.000,B 0.000,C 90.000,E1 109.214} C_DIS
LIN {X -0.081,Y -409.160,Z 1130.594,A 0.000,B 0.000,C 90.000,E1 106.985} C_DIS
LIN {X 0.029,Y -427.187,Z 1130.582,A 0.000,B 0.000,C 90.000,E1 104.773} C_DIS
LIN {X 0.073,Y -446.768,Z 1130.570,A 0.000,B 0.000,C 90.000,E1 102.647} C_DIS
LIN {X -0.193,Y -469.470,Z 1130.558,A 0.000,B 0.000,C 90.000,E1 100.489} C_DIS
LIN {X -0.163,Y -471.313,Z 1130.557,A 0.000,B 0.000,C 90.000,E1 100.254} C_DIS
LIN {X 0.156,Y -472.838,Z 1130.555,A 0.000,B 0.000,C 90.000,E1 99.962} C_DIS
LIN {X 0.009,Y -473.980,Z 1130.554,A 0.000,B 0.000,C 90.000,E1 99.726} C_DIS
LIN {X 0.122,Y -475.347,Z 1130.551,A 0.000,B 0.000,C 90.000,E1 99.208} C_DIS
LIN {X -0.225,Y -475.690,Z 1130.548,A 0.000,B 0.000,C 90.000,E1 98.746} C_DIS
LIN {X -0.023,Y -475.070,Z 1130.546,A 0.000,B 0.000,C 90.000,E1 98.219} C_DIS
LIN {X 0.111,Y -473.387,Z 1130.543,A 0.000,B 0.000,C 90.000,E1 97.701} C_DIS
LIN {X -0.028,Y -472.054,Z 1130.542,A 0.000,B 0.000,C 90.000,E1 97.466} C_DIS
LIN {X 0.103,Y -455.850,Z 1130.529,A 0.000,B 0.000,C 90.000,E1 95.163} C_DIS
LIN {X 0.045,Y -441.687,Z 1130.517,A 0.000,B 0.000,C 90.000,E1 93.094} C_DIS
LIN {X 0.038,Y -423.762,Z 1130.501,A 0.000,B 0.000,C 90.000,E1 90.172} C_DIS
LIN {X -0.094,Y -407.316,Z 1130.484,A 0.000,B 0.000,C 90.000,E1 87.192} C_DIS
LIN {X -0.102,Y -398.333,Z 1130.475,A 0.000,B 0.000,C 90.000,E1 85.527} C_DIS
LIN {X -0.179,Y -386.405,Z 1130.463,A 0.000,B 0.000,C 90.000,E1 83.280} C_DIS
LIN {X -0.089,Y -377.384,Z 1130.453,A 0.000,B 0.000,C 90.000,E1 81.546} C_DIS
LIN {X -0.107,Y -368.190,Z 1130.443,A 0.000,B 0.000,C 90.000,E1 79.803} C_DIS
LIN {X 0.160,Y -360.207,Z 1130.435,A 0.000,B 0.000,C 90.000,E1 78.285} C_DIS
LIN {X -0.086,Y -348.745,Z 1130.423,A 0.000,B 0.000,C 90.000,E1 76.228} C_DIS
LIN {X -0.152,Y -337.239,Z 1130.411,A 0.000,B 0.000,C 90.000,E1 74.102} C_DIS
LIN {X -0.047,Y -322.758,Z 1130.396,A 0.000,B 0.000,C 90.000,E1 71.275} C_DIS
LIN {X -0.132,Y -309.203,Z 1130.380,A 0.000,B 0.000,C 90.000,E1 68.411} C_DIS
LIN {X 0.033,Y -296.426,Z 1130.364,A 0.000,B 0.000,C 90.000,E1 65.433} C_DIS
LIN {X 0.065,Y -284.121,Z 1130.347,A 0.000,B 0.000,C 90.000,E1 62.410} C_DIS
LIN {X 0.034,Y -272.317,Z 1130.330,A 0.000,B 0.000,C 90.000,E1 59.331} C_DIS
LIN {X -0.045,Y -262.272,Z 1130.314,A 0.000,B 0.000,C 90.000,E1 56.548} C_DIS
LIN {X -0.055,Y -251.456,Z 1130.296,A 0.000,B 0.000,C 90.000,E1 53.336} C_DIS
LIN {X -0.119,Y -241.344,Z 1130.278,A 0.000,B 0.000,C 90.000,E1 50.070} C_DIS
LIN {X 0.033,Y -233.167,Z 1130.261,A 0.000,B 0.000,C 90.000,E1 47.067} C_DIS
LIN {X -0.007,Y -223.460,Z 1130.240,A 0.000,B 0.000,C 90.000,E1 43.299} C_DIS
LIN {X 0.014,Y -216.161,Z 1130.223,A 0.000,B 0.000,C 90.000,E1 40.216} C_DIS
LIN {X 0.069,Y -209.223,Z 1130.206,A 0.000,B 0.000,C 90.000,E1 37.076} C_DIS
LIN {X 0.040,Y -202.708,Z 1130.188,A 0.000,B 0.000,C 90.000,E1 33.913} C_DIS
LIN {X 0.082,Y -195.376,Z 1130.166,A 0.000,B 0.000,C 90.000,E1 29.873} C_DIS
LIN {X 0.042,Y -190.182,Z 1130.148,A 0.000,B 0.000,C 90.000,E1 26.616} C_DIS
LIN {X -0.035,Y -185.626,Z 1130.130,A 0.000,B 0.000,C 90.000,E1 23.334} C_DIS
LIN {X 0.009,Y -180.810,Z 1130.106,A 0.000,B 0.000,C 90.000,E1 19.141} C_DIS
LIN {X 0.069,Y -176.992,Z 1130.083,A 0.000,B 0.000,C 90.000,E1 14.898} C_DIS
LIN {X 0.010,Y -174.231,Z 1130.059,A 0.000,B 0.000,C 90.000,E1 10.658} C_DIS
LIN {X 0.045,Y -171.954,Z 1130.021,A 0.000,B 0.000,C 90.000,E1 3.784} C_DIS
LIN {X -0.014,Y -173.428,Z 1129.964,A 0.000,B 0.000,C 90.000,E1 353.514} C_DIS
LIN {X 0.092,Y -176.314,Z 1129.935,A 0.000,B 0.000,C 90.000,E1 348.342} C_DIS
LIN {X 0.051,Y -179.764,Z 1129.912,A 0.000,B 0.000,C 90.000,E1 344.102} C_DIS
LIN {X 0.066,Y -184.009,Z 1129.888,A 0.000,B 0.000,C 90.000,E1 339.880} C_DIS
LIN {X 0.060,Y -188.122,Z 1129.870,A 0.000,B 0.000,C 90.000,E1 336.538} C_DIS
LIN {X -0.039,Y -192.875,Z 1129.851,A 0.000,B 0.000,C 90.000,E1 333.256} C_DIS
LIN {X -0.111,Y -198.294,Z 1129.833,A 0.000,B 0.000,C 90.000,E1 329.999} C_DIS
LIN {X 0.082,Y -204.232,Z 1129.815,A 0.000,B 0.000,C 90.000,E1 326.707} C_DIS
LIN {X -0.024,Y -211.041,Z 1129.797,A 0.000,B 0.000,C 90.000,E1 323.543} C_DIS
LIN {X 0.040,Y -219.618,Z 1129.778,A 0.000,B 0.000,C 90.000,E1 319.989} C_DIS
LIN {X 0.044,Y -228.203,Z 1129.761,A 0.000,B 0.000,C 90.000,E1 316.905} C_DIS
LIN {X 0.101,Y -237.785,Z 1129.744,A 0.000,B 0.000,C 90.000,E1 313.866} C_DIS
LIN {X -0.072,Y -245.735,Z 1129.731,A 0.000,B 0.000,C 90.000,E1 311.676} C_DIS
LIN {X -0.062,Y -255.963,Z 1129.717,A 0.000,B 0.000,C 90.000,E1 309.116} C_DIS
LIN {X 0.130,Y -269.086,Z 1129.701,A 0.000,B 0.000,C 90.000,E1 306.217} C_DIS
LIN {X 0.156,Y -285.252,Z 1129.684,A 0.000,B 0.000,C 90.000,E1 303.086} C_DIS
LIN {X 0.019,Y -296.849,Z 1129.673,A 0.000,B 0.000,C 90.000,E1 301.082} C_DIS
LIN {X 0.083,Y -316.080,Z 1129.656,A 0.000,B 0.000,C 90.000,E1 298.103} C_DIS
LIN {X -0.106,Y -332.269,Z 1129.644,A 0.000,B 0.000,C 90.000,E1 295.899} C_DIS
LIN {X -0.016,Y -347.404,Z 1129.633,A 0.000,B 0.000,C 90.000,E1 294.027} C_DIS
LIN {X -0.105,Y -363.215,Z 1129.624,A 0.000,B 0.000,C 90.000,E1 292.333} C_DIS
LIN {X 0.151,Y -390.284,Z 1129.610,A 0.000,B 0.000,C 90.000,E1 289.758} C_DIS
LIN {X 0.189,Y -403.835,Z 1129.603,A 0.000,B 0.000,C 90.000,E1 288.544} C_DIS
LIN {X 0.025,Y -414.351,Z 1129.598,A 0.000,B 0.000,C 90.000,E1 287.583} C_DIS
LIN {X -0.219,Y -422.081,Z 1129.594,A 0.000,B 0.000,C 90.000,E1 286.858} C_DIS
LIN {X -0.190,Y -429.590,Z 1129.589,A 0.000,B 0.000,C 90.000,E1 286.079} C_DIS
LIN {X 0.101,Y -436.849,Z 1129.585,A 0.000,B 0.000,C 90.000,E1 285.245} C_DIS
LIN {X -0.160,Y -443.709,Z 1129.580,A 0.000,B 0.000,C 90.000,E1 284.481} C_DIS
LIN {X 0.190,Y -449.894,Z 1129.576,A 0.000,B 0.000,C 90.000,E1 283.647} C_DIS
LIN {X 0.045,Y -455.403,Z 1129.572,A 0.000,B 0.000,C 90.000,E1 282.883} C_DIS
LIN {X -0.048,Y -460.156,Z 1129.567,A 0.000,B 0.000,C 90.000,E1 282.119} C_DIS
LIN {X -0.198,Y -464.264,Z 1129.563,A 0.000,B 0.000,C 90.000,E1 281.366} C_DIS
LIN {X -0.215,Y -467.851,Z 1129.559,A 0.000,B 0.000,C 90.000,E1 280.602} C_DIS
LIN {X 0.172,Y -470.985,Z 1129.555,A 0.000,B 0.000,C 90.000,E1 279.792} C_DIS
LIN {X -0.124,Y -472.738,Z 1129.552,A 0.000,B 0.000,C 90.000,E1 279.321} C_DIS
LIN {X -0.020,Y -474.248,Z 1129.549,A 0.000,B 0.000,C 90.000,E1 278.803} C_DIS
LIN {X 0.166,Y -475.406,Z 1129.546,A 0.000,B 0.000,C 90.000,E1 278.276} C_DIS
LIN {X -0.180,Y -476.318,Z 1129.543,A 0.000,B 0.000,C 90.000,E1 277.814} C_DIS
LIN {X -0.047,Y -476.938,Z 1129.541,A 0.000,B 0.000,C 90.000,E1 277.296} C_DIS
LIN {X 0.093,Y -477.205,Z 1129.538,A 0.000,B 0.000,C 90.000,E1 276.777} C_DIS
LIN {X 0.237,Y -477.107,Z 1129.535,A 0.000,B 0.000,C 90.000,E1 276.258} C_DIS
LIN {X -0.092,Y -476.726,Z 1129.532,A 0.000,B 0.000,C 90.000,E1 275.796} C_DIS
LIN {X 0.051,Y -475.992,Z 1129.529,A 0.000,B 0.000,C 90.000,E1 275.277} C_DIS
LIN {X 0.191,Y -474.887,Z 1129.527,A 0.000,B 0.000,C 90.000,E1 274.759} C_DIS
LIN {X -0.184,Y -473.378,Z 1129.524,A 0.000,B 0.000,C 90.000,E1 274.302} C_DIS
LIN {X -0.056,Y -471.361,Z 1129.521,A 0.000,B 0.000,C 90.000,E1 273.784} C_DIS
LIN {X 0.032,Y -468.690,Z 1129.518,A 0.000,B 0.000,C 90.000,E1 273.269} C_DIS
LIN {X -0.140,Y -467.070,Z 1129.517,A 0.000,B 0.000,C 90.000,E1 273.037} C_DIS
LIN {X -0.077,Y -463.078,Z 1129.514,A 0.000,B 0.000,C 90.000,E1 272.522} C_DIS
LIN {X 0.024,Y -457.835,Z 1129.511,A 0.000,B 0.000,C 90.000,E1 272.007} C_DIS
LIN {X -0.118,Y -454.759,Z 1129.510,A 0.000,B 0.000,C 90.000,E1 271.776} C_DIS
LIN {X 0.065,Y -448.251,Z 1129.507,A 0.000,B 0.000,C 90.000,E1 271.318} C_DIS
LIN {X -0.092,Y -441.530,Z 1129.505,A 0.000,B 0.000,C 90.000,E1 270.974} C_DIS
LIN {X 0.185,Y -434.459,Z 1129.504,A 0.000,B 0.000,C 90.000,E1 270.630} C_DIS
LIN {X -0.052,Y -427.295,Z 1129.502,A 0.000,B 0.000,C 90.000,E1 270.401} C_DIS
LIN {X 0.032,Y -419.910,Z 1129.501,A 0.000,B 0.000,C 90.000,E1 270.172} C_DIS
LIN {X 0.011,Y -412.529,Z 1129.500,A 0.000,B 0.000,C 90.000,E1 270.000} C_DIS
LIN {X -0.198,Y -401.394,Z 1129.499,A 0.000,B 0.000,C 90.000,E1 269.828} C_DIS
LIN {X 0.105,Y -389.315,Z 1129.498,A 0.000,B 0.000,C 90.000,E1 269.656} C_DIS
LIN {X -0.099,Y -380.843,Z 1129.498,A 0.000,B 0.000,C 90.000,E1 269.656} C_DIS
LIN {X -0.070,Y -181.474,Z 1129.498,A 0.000,B 0.000,C 90.000,E1 269.656} C_DIS
LIN {X 0.074,Y -180.906,Z 1129.474,A 0.000,B 0.000,C 90.000,E1 265.355} C_DIS
LIN {X -0.032,Y -180.693,Z 1129.470,A 0.000,B 0.000,C 90.000,E1 264.546} C_DIS
LIN {X 0.046,Y -178.778,Z 1129.442,A 0.000,B 0.000,C 90.000,E1 259.454} C_DIS
LIN {X -0.052,Y -175.825,Z 1129.413,A 0.000,B 0.000,C 90.000,E1 254.393} C_DIS
LIN {X -0.051,Y -172.012,Z 1129.385,A 0.000,B 0.000,C 90.000,E1 249.263} C_DIS
LIN {X -0.074,Y -171.432,Z 1129.380,A 0.000,B 0.000,C 90.000,E1 248.411} C_DIS
LIN {X -0.019,Y -167.668,Z 1129.356,A 0.000,B 0.000,C 90.000,E1 244.076} C_DIS
LIN {X -0.079,Y -166.341,Z 1129.346,A 0.000,B 0.000,C 90.000,E1 242.359} C_DIS
LIN {X -0.086,Y -163.078,Z 1129.327,A 0.000,B 0.000,C 90.000,E1 238.869} C_DIS
LIN {X -0.035,Y -161.018,Z 1129.312,A 0.000,B 0.000,C 90.000,E1 236.215} C_DIS
LIN {X -0.050,Y -157.760,Z 1129.293,A 0.000,B 0.000,C 90.000,E1 232.683} C_DIS
LIN {X 0.013,Y -155.799,Z 1129.278,A 0.000,B 0.000,C 90.000,E1 229.989} C_DIS
LIN {X 0.067,Y -152.051,Z 1129.253,A 0.000,B 0.000,C 90.000,E1 225.486} C_DIS
LIN {X 0.084,Y -150.300,Z 1129.238,A 0.000,B 0.000,C 90.000,E1 222.771} C_DIS
LIN {X 0.009,Y -147.046,Z 1129.213,A 0.000,B 0.000,C 90.000,E1 218.257} C_DIS
LIN {X 0.002,Y -145.625,Z 1129.197,A 0.000,B 0.000,C 90.000,E1 215.518} C_DIS
LIN {X 0.001,Y -143.009,Z 1129.172,A 0.000,B 0.000,C 90.000,E1 210.924} C_DIS
LIN {X -0.068,Y -141.636,Z 1129.151,A 0.000,B 0.000,C 90.000,E1 207.257} C_DIS
LIN {X -0.017,Y -139.437,Z 1129.115,A 0.000,B 0.000,C 90.000,E1 200.737} C_DIS
LIN {X 0.037,Y -139.169,Z 1129.105,A 0.000,B 0.000,C 90.000,E1 198.852} C_DIS
LIN {X -0.066,Y -138.317,Z 1129.053,A 0.000,B 0.000,C 90.000,E1 189.557} C_DIS
LIN {X -0.057,Y -139.474,Z 1129.006,A 0.000,B 0.000,C 90.000,E1 181.146} C_DIS
LIN {X 0.024,Y -141.051,Z 1128.975,A 0.000,B 0.000,C 90.000,E1 175.527} C_DIS
LIN {X -0.022,Y -142.422,Z 1128.960,A 0.000,B 0.000,C 90.000,E1 172.761} C_DIS
LIN {X 0.038,Y -144.658,Z 1128.934,A 0.000,B 0.000,C 90.000,E1 168.117} C_DIS
LIN {X 0.022,Y -147.241,Z 1128.914,A 0.000,B 0.000,C 90.000,E1 164.448} C_DIS
LIN {X 0.041,Y -150.557,Z 1128.888,A 0.000,B 0.000,C 90.000,E1 159.880} C_DIS
LIN {X -0.020,Y -154.025,Z 1128.868,A 0.000,B 0.000,C 90.000,E1 156.282} C_DIS
LIN {X 0.048,Y -157.440,Z 1128.848,A 0.000,B 0.000,C 90.000,E1 152.666} C_DIS
LIN {X -0.002,Y -161.656,Z 1128.828,A 0.000,B 0.000,C 90.000,E1 149.125} C_DIS
LIN {X 0.015,Y -165.851,Z 1128.809,A 0.000,B 0.000,C 90.000,E1 145.595} C_DIS
LIN {X 0.007,Y -170.826,Z 1128.790,A 0.000,B 0.000,C 90.000,E1 142.110} C_DIS
LIN {X -0.078,Y -175.695,Z 1128.770,A 0.000,B 0.000,C 90.000,E1 138.690} C_DIS
LIN {X 0.046,Y -181.308,Z 1128.751,A 0.000,B 0.000,C 90.000,E1 135.243} C_DIS
LIN {X -0.082,Y -186.789,Z 1128.733,A 0.000,B 0.000,C 90.000,E1 131.919} C_DIS
LIN {X -0.012,Y -191.382,Z 1128.719,A 0.000,B 0.000,C 90.000,E1 129.402} C_DIS
LIN {X 0.071,Y -197.224,Z 1128.701,A 0.000,B 0.000,C 90.000,E1 126.091} C_DIS
LIN {X 0.019,Y -200.875,Z 1128.690,A 0.000,B 0.000,C 90.000,E1 124.278} C_DIS
LIN {X -0.007,Y -309.296,Z 1128.690,A 0.000,B 0.000,C 90.000,E1 124.278} C_DIS
LIN {X 0.161,Y -312.045,Z 1128.690,A 0.000,B 0.000,C 90.000,E1 124.199} C_DIS
LIN {X 0.213,Y -317.071,Z 1128.689,A 0.000,B 0.000,C 90.000,E1 123.913} C_DIS
LIN {X 0.087,Y -319.870,Z 1128.687,A 0.000,B 0.000,C 90.000,E1 123.658} C_DIS
LIN {X 0.184,Y -323.537,Z 1128.684,A 0.000,B 0.000,C 90.000,E1 123.086} C_DIS
LIN {X -0.007,Y -325.008,Z 1128.682,A 0.000,B 0.000,C 90.000,E1 122.801} C_DIS
LIN {X -0.092,Y -336.959,Z 1128.665,A 0.000,B 0.000,C 90.000,E1 119.667} C_DIS
LIN {X 0.012,Y -349.107,Z 1128.649,A 0.000,B 0.000,C 90.000,E1 116.873} C_DIS
LIN {X 0.011,Y -362.730,Z 1128.634,A 0.000,B 0.000,C 90.000,E1 114.155} C_DIS
LIN {X 0.142,Y -376.180,Z 1128.621,A 0.000,B 0.000,C 90.000,E1 111.770} C_DIS
LIN {X 0.190,Y -390.986,Z 1128.608,A 0.000,B 0.000,C 90.000,E1 109.450} C_DIS
LIN {X -0.020,Y -407.256,Z 1128.596,A 0.000,B 0.000,C 90.000,E1 107.221} C_DIS
LIN {X 0.043,Y -425.102,Z 1128.583,A 0.000,B 0.000,C 90.000,E1 105.009} C_DIS
LIN {X -0.006,Y -444.542,Z 1128.572,A 0.000,B 0.000,C 90.000,E1 102.883} C_DIS
LIN {X 0.088,Y -464.773,Z 1128.561,A 0.000,B 0.000,C 90.000,E1 100.894} C_DIS
LIN {X 0.030,Y -469.698,Z 1128.558,A 0.000,B 0.000,C 90.000,E1 100.433} C_DIS
LIN {X 0.063,Y -471.473,Z 1128.557,A 0.000,B 0.000,C 90.000,E1 100.197} C_DIS
LIN {X -0.082,Y -472.947,Z 1128.555,A 0.000,B 0.000,C 90.000,E1 99.962} C_DIS
LIN {X 0.238,Y -474.047,Z 1128.554,A 0.000,B 0.000,C 90.000,E1 99.670} C_DIS
LIN {X -0.116,Y -475.348,Z 1128.551,A 0.000,B 0.000,C 90.000,E1 99.208} C_DIS
LIN {X 0.080,Y -475.635,Z 1128.548,A 0.000,B 0.000,C 90.000,E1 98.681} C_DIS
LIN {X 0.210,Y -474.954,Z 1128.546,A 0.000,B 0.000,C 90.000,E1 98.163} C_DIS
LIN {X -0.126,Y -473.202,Z 1128.543,A 0.000,B 0.000,C 90.000,E1 97.701} C_DIS
LIN {X 0.204,Y -471.823,Z 1128.541,A 0.000,B 0.000,C 90.000,E1 97.409} C_DIS
LIN {X -0.131,Y -455.597,Z 1128.529,A 0.000,B 0.000,C 90.000,E1 95.163} C_DIS
LIN {X -0.188,Y -441.440,Z 1128.517,A 0.000,B 0.000,C 90.000,E1 93.094} C_DIS
LIN {X 0.103,Y -425.114,Z 1128.502,A 0.000,B 0.000,C 90.000,E1 90.401} C_DIS
LIN {X 0.008,Y -408.560,Z 1128.486,A 0.000,B 0.000,C 90.000,E1 87.421} C_DIS
LIN {X 0.021,Y -399.604,Z 1128.476,A 0.000,B 0.000,C 90.000,E1 85.755} C_DIS
LIN {X -0.068,Y -387.648,Z 1128.464,A 0.000,B 0.000,C 90.000,E1 83.514} C_DIS
LIN {X 0.058,Y -377.133,Z 1128.453,A 0.000,B 0.000,C 90.000,E1 81.489} C_DIS
LIN {X 0.033,Y -369.478,Z 1128.445,A 0.000,B 0.000,C 90.000,E1 80.038} C_DIS
LIN {X -0.035,Y -361.531,Z 1128.437,A 0.000,B 0.000,C 90.000,E1 78.578} C_DIS
LIN {X 0.089,Y -350.085,Z 1128.425,A 0.000,B 0.000,C 90.000,E1 76.464} C_DIS
LIN {X 0.050,Y -338.585,Z 1128.413,A 0.000,B 0.000,C 90.000,E1 74.338} C_DIS
LIN {X 0.078,Y -324.050,Z 1128.397,A 0.000,B 0.000,C 90.000,E1 71.529} C_DIS
LIN {X 0.050,Y -308.927,Z 1128.380,A 0.000,B 0.000,C 90.000,E1 68.337} C_DIS
LIN {X -0.061,Y -296.150,Z 1128.363,A 0.000,B 0.000,C 90.000,E1 65.409} C_DIS
LIN {X -0.125,Y -285.196,Z 1128.348,A 0.000,B 0.000,C 90.000,E1 62.743} C_DIS
LIN {X -0.068,Y -274.634,Z 1128.333,A 0.000,B 0.000,C 90.000,E1 59.999} C_DIS
LIN {X 0.048,Y -263.203,Z 1128.316,A 0.000,B 0.000,C 90.000,E1 56.834} C_DIS
LIN {X 0.060,Y -252.346,Z 1128.298,A 0.000,B 0.000,C 90.000,E1 53.623} C_DIS
LIN {X 0.018,Y -243.179,Z 1128.282,A 0.000,B 0.000,C 90.000,E1 50.723} C_DIS
LIN {X -0.009,Y -232.855,Z 1128.261,A 0.000,B 0.000,C 90.000,E1 47.025} C_DIS
LIN {X -0.057,Y -223.122,Z 1128.240,A 0.000,B 0.000,C 90.000,E1 43.257} C_DIS
LIN {X -0.036,Y -215.809,Z 1128.223,A 0.000,B 0.000,C 90.000,E1 40.172} C_DIS
LIN {X -0.014,Y -207.180,Z 1128.201,A 0.000,B 0.000,C 90.000,E1 36.251} C_DIS
LIN {X -0.087,Y -200.817,Z 1128.184,A 0.000,B 0.000,C 90.000,E1 33.086} C_DIS
LIN {X 0.030,Y -195.000,Z 1128.166,A 0.000,B 0.000,C 90.000,E1 29.823} C_DIS
LIN {X -0.013,Y -189.811,Z 1128.148,A 0.000,B 0.000,C 90.000,E1 26.565} C_DIS
LIN {X -0.019,Y -185.251,Z 1128.129,A 0.000,B 0.000,C 90.000,E1 23.259} C_DIS
LIN {X -0.054,Y -180.452,Z 1128.106,A 0.000,B 0.000,C 90.000,E1 19.087} C_DIS
LIN {X 0.046,Y -176.652,Z 1128.083,A 0.000,B 0.000,C 90.000,E1 14.828} C_DIS
LIN {X -0.064,Y -173.911,Z 1128.059,A 0.000,B 0.000,C 90.000,E1 10.602} C_DIS
LIN {X -0.041,Y -171.663,Z 1128.021,A 0.000,B 0.000,C 90.000,E1 3.726} C_DIS
LIN {X -0.026,Y -173.128,Z 1127.964,A 0.000,B 0.000,C 90.000,E1 353.514} C_DIS
LIN {X 0.068,Y -175.981,Z 1127.935,A 0.000,B 0.000,C 90.000,E1 348.342} C_DIS
LIN {X 0.017,Y -179.420,Z 1127.912,A 0.000,B 0.000,C 90.000,E1 344.102} C_DIS
LIN {X 0.020,Y -183.672,Z 1127.888,A 0.000,B 0.000,C 90.000,E1 339.880} C_DIS
LIN {X 0.004,Y -187.775,Z 1127.870,A 0.000,B 0.000,C 90.000,E1 336.538} C_DIS
LIN {X -0.105,Y -192.542,Z 1127.851,A 0.000,B 0.000,C 90.000,E1 333.256} C_DIS
LIN {X -0.015,Y -197.980,Z 1127.833,A 0.000,B 0.000,C 90.000,E1 329.950} C_DIS
LIN {X -0.004,Y -203.947,Z 1127.815,A 0.000,B 0.000,C 90.000,E1 326.707} C_DIS
LIN {X 0.048,Y -210.798,Z 1127.797,A 0.000,B 0.000,C 90.000,E1 323.497} C_DIS
LIN {X 0.020,Y -218.383,Z 1127.780,A 0.000,B 0.000,C 90.000,E1 320.356} C_DIS
LIN {X 0.003,Y -226.871,Z 1127.763,A 0.000,B 0.000,C 90.000,E1 317.268} C_DIS
LIN {X -0.152,Y -236.352,Z 1127.746,A 0.000,B 0.000,C 90.000,E1 314.271} C_DIS
LIN {X -0.014,Y -244.190,Z 1127.733,A 0.000,B 0.000,C 90.000,E1 312.000} C_DIS
LIN {X -0.008,Y -255.863,Z 1127.717,A 0.000,B 0.000,C 90.000,E1 309.072} C_DIS
LIN {X -0.024,Y -269.061,Z 1127.701,A 0.000,B 0.000,C 90.000,E1 306.217} C_DIS
LIN {X -0.007,Y -285.285,Z 1127.684,A 0.000,B 0.000,C 90.000,E1 303.086} C_DIS
LIN {X 0.002,Y -296.905,Z 1127.672,A 0.000,B 0.000,C 90.000,E1 301.052} C_DIS
LIN {X -0.096,Y -316.191,Z 1127.656,A 0.000,B 0.000,C 90.000,E1 298.103} C_DIS
LIN {X 0.009,Y -332.416,Z 1127.644,A 0.000,B 0.000,C 90.000,E1 295.848} C_DIS
LIN {X -0.062,Y -347.562,Z 1127.633,A 0.000,B 0.000,C 90.000,E1 294.003} C_DIS
LIN {X -0.085,Y -363.574,Z 1127.624,A 0.000,B 0.000,C 90.000,E1 292.280} C_DIS
LIN {X 0.117,Y -390.791,Z 1127.610,A 0.000,B 0.000,C 90.000,E1 289.704} C_DIS
LIN {X -0.188,Y -404.310,Z 1127.603,A 0.000,B 0.000,C 90.000,E1 288.544} C_DIS
LIN {X 0.179,Y -414.820,Z 1127.597,A 0.000,B 0.000,C 90.000,E1 287.511} C_DIS
LIN {X -0.182,Y -422.575,Z 1127.593,A 0.000,B 0.000,C 90.000,E1 286.804} C_DIS
LIN {X -0.162,Y -430.078,Z 1127.589,A 0.000,B 0.000,C 90.000,E1 286.024} C_DIS
LIN {X 0.127,Y -437.363,Z 1127.584,A 0.000,B 0.000,C 90.000,E1 285.190} C_DIS
LIN {X -0.016,Y -444.165,Z 1127.580,A 0.000,B 0.000,C 90.000,E1 284.411} C_DIS
LIN {X 0.229,Y -450.361,Z 1127.576,A 0.000,B 0.000,C 90.000,E1 283.592} C_DIS
LIN {X 0.091,Y -455.834,Z 1127.571,A 0.000,B 0.000,C 90.000,E1 282.827} C_DIS
LIN {X 0.003,Y -460.596,Z 1127.567,A 0.000,B 0.000,C 90.000,E1 282.063} C_DIS
LIN {X -0.049,Y -464.698,Z 1127.563,A 0.000,B 0.000,C 90.000,E1 281.299} C_DIS
LIN {X -0.153,Y -468.286,Z 1127.558,A 0.000,B 0.000,C 90.000,E1 280.546} C_DIS
LIN {X -0.144,Y -471.395,Z 1127.554,A 0.000,B 0.000,C 90.000,E1 279.782} C_DIS
LIN {X -0.054,Y -473.146,Z 1127.551,A 0.000,B 0.000,C 90.000,E1 279.265} C_DIS
LIN {X 0.054,Y -474.594,Z 1127.549,A 0.000,B 0.000,C 90.000,E1 278.746} C_DIS
LIN {X 0.243,Y -475.735,Z 1127.546,A 0.000,B 0.000,C 90.000,E1 278.219} C_DIS
LIN {X -0.101,Y -476.618,Z 1127.543,A 0.000,B 0.000,C 90.000,E1 277.757} C_DIS
LIN {X 0.035,Y -477.195,Z 1127.540,A 0.000,B 0.000,C 90.000,E1 277.239} C_DIS
LIN {X 0.178,Y -477.427,Z 1127.537,A 0.000,B 0.000,C 90.000,E1 276.720} C_DIS
LIN {X -0.151,Y -477.365,Z 1127.535,A 0.000,B 0.000,C 90.000,E1 276.258} C_DIS
LIN {X -0.004,Y -476.981,Z 1127.532,A 0.000,B 0.000,C 90.000,E1 275.739} C_DIS
LIN {X 0.142,Y -476.212,Z 1127.529,A 0.000,B 0.000,C 90.000,E1 275.220} C_DIS
LIN {X -0.191,Y -475.136,Z 1127.526,A 0.000,B 0.000,C 90.000,E1 274.759} C_DIS
LIN {X -0.092,Y -473.612,Z 1127.524,A 0.000,B 0.000,C 90.000,E1 274.245} C_DIS
LIN {X 0.038,Y -471.553,Z 1127.521,A 0.000,B 0.000,C 90.000,E1 273.726} C_DIS
LIN {X 0.127,Y -468.866,Z 1127.518,A 0.000,B 0.000,C 90.000,E1 273.212} C_DIS
LIN {X 0.223,Y -465.306,Z 1127.515,A 0.000,B 0.000,C 90.000,E1 272.694} C_DIS
LIN {X 0.018,Y -463.167,Z 1127.514,A 0.000,B 0.000,C 90.000,E1 272.465} C_DIS
LIN {X 0.114,Y -457.873,Z 1127.511,A 0.000,B 0.000,C 90.000,E1 271.949} C_DIS
LIN {X -0.034,Y -454.754,Z 1127.510,A 0.000,B 0.000,C 90.000,E1 271.718} C_DIS
LIN {X 0.174,Y -448.247,Z 1127.507,A 0.000,B 0.000,C 90.000,E1 271.260} C_DIS
LIN {X 0.039,Y -441.446,Z 1127.505,A 0.000,B 0.000,C 90.000,E1 270.917} C_DIS
LIN {X -0.077,Y -434.458,Z 1127.503,A 0.000,B 0.000,C 90.000,E1 270.630} C_DIS
LIN {X 0.133,Y -427.262,Z 1127.502,A 0.000,B 0.000,C 90.000,E1 270.344} C_DIS
LIN {X -0.170,Y -419.974,Z 1127.501,A 0.000,B 0.000,C 90.000,E1 270.172} C_DIS
LIN {X -0.182,Y -412.621,Z 1127.500,A 0.000,B 0.000,C 90.000,E1 270.000} C_DIS
LIN {X 0.020,Y -401.365,Z 1127.499,A 0.000,B 0.000,C 90.000,E1 269.771} C_DIS
LIN {X 0.096,Y -391.611,Z 1127.498,A 0.000,B 0.000,C 90.000,E1 269.656} C_DIS
LIN {X 0.175,Y -380.752,Z 1127.498,A 0.000,B 0.000,C 90.000,E1 269.599} C_DIS
LIN {X 0.064,Y -181.469,Z 1127.498,A 0.000,B 0.000,C 90.000,E1 269.599} C_DIS
LIN {X 0.027,Y -180.906,Z 1127.474,A 0.000,B 0.000,C 90.000,E1 265.355} C_DIS
LIN {X -0.079,Y -180.686,Z 1127.470,A 0.000,B 0.000,C 90.000,E1 264.546} C_DIS
LIN {X -0.001,Y -178.770,Z 1127.441,A 0.000,B 0.000,C 90.000,E1 259.454} C_DIS
LIN {X 0.072,Y -175.817,Z 1127.413,A 0.000,B 0.000,C 90.000,E1 254.338} C_DIS
LIN {X 0.065,Y -172.003,Z 1127.385,A 0.000,B 0.000,C 90.000,E1 249.209} C_DIS
LIN {X 0.040,Y -171.419,Z 1127.380,A 0.000,B 0.000,C 90.000,E1 248.358} C_DIS
LIN {X 0.086,Y -167.658,Z 1127.356,A 0.000,B 0.000,C 90.000,E1 244.024} C_DIS
LIN {X 0.024,Y -166.325,Z 1127.346,A 0.000,B 0.000,C 90.000,E1 242.308} C_DIS
LIN {X 0.010,Y -163.065,Z 1127.327,A 0.000,B 0.000,C 90.000,E1 238.820} C_DIS
LIN {X -0.078,Y -161.003,Z 1127.312,A 0.000,B 0.000,C 90.000,E1 236.215} C_DIS
LIN {X 0.032,Y -157.748,Z 1127.292,A 0.000,B 0.000,C 90.000,E1 232.637} C_DIS
LIN {X -0.030,Y -155.786,Z 1127.278,A 0.000,B 0.000,C 90.000,E1 229.989} C_DIS
LIN {X 0.025,Y -152.039,Z 1127.253,A 0.000,B 0.000,C 90.000,E1 225.486} C_DIS
LIN {X 0.043,Y -150.289,Z 1127.238,A 0.000,B 0.000,C 90.000,E1 222.771} C_DIS
LIN {X -0.032,Y -147.037,Z 1127.213,A 0.000,B 0.000,C 90.000,E1 218.257} C_DIS
LIN {X -0.038,Y -145.617,Z 1127.197,A 0.000,B 0.000,C 90.000,E1 215.518} C_DIS
LIN {X -0.039,Y -143.002,Z 1127.172,A 0.000,B 0.000,C 90.000,E1 210.924} C_DIS
LIN {X 0.018,Y -141.629,Z 1127.151,A 0.000,B 0.000,C 90.000,E1 207.206} C_DIS
LIN {X -0.057,Y -139.434,Z 1127.115,A 0.000,B 0.000,C 90.000,E1 200.737} C_DIS
LIN {X -0.003,Y -139.165,Z 1127.105,A 0.000,B 0.000,C 90.000,E1 198.852} C_DIS
LIN {X 0.031,Y -138.316,Z 1127.053,A 0.000,B 0.000,C 90.000,E1 189.500} C_DIS
LIN {X 0.042,Y -139.476,Z 1127.006,A 0.000,B 0.000,C 90.000,E1 181.088} C_DIS
LIN {X -0.017,Y -141.058,Z 1126.975,A 0.000,B 0.000,C 90.000,E1 175.527} C_DIS
LIN {X -0.063,Y -142.430,Z 1126.960,A 0.000,B 0.000,C 90.000,E1 172.761} C_DIS
LIN {X -0.003,Y -144.668,Z 1126.934,A 0.000,B 0.000,C 90.000,E1 168.117} C_DIS
LIN {X -0.019,Y -147.253,Z 1126.914,A 0.000,B 0.000,C 90.000,E1 164.448} C_DIS
LIN {X -0.001,Y -150.570,Z 1126.888,A 0.000,B 0.000,C 90.000,E1 159.880} C_DIS
LIN {X 0.078,Y -154.040,Z 1126.868,A 0.000,B 0.000,C 90.000,E1 156.230} C_DIS
LIN {X 0.005,Y -157.457,Z 1126.848,A 0.000,B 0.000,C 90.000,E1 152.666} C_DIS
LIN {X -0.046,Y -161.676,Z 1126.828,A 0.000,B 0.000,C 90.000,E1 149.125} C_DIS
LIN {X -0.029,Y -165.871,Z 1126.809,A 0.000,B 0.000,C 90.000,E1 145.595} C_DIS
LIN {X -0.038,Y -170.849,Z 1126.789,A 0.000,B 0.000,C 90.000,E1 142.110} C_DIS
LIN {X 0.008,Y -175.718,Z 1126.770,A 0.000,B 0.000,C 90.000,E1 138.647} C_DIS
LIN {X -0.001,Y -181.330,Z 1126.751,A 0.000,B 0.000,C 90.000,E1 135.243} C_DIS
LIN {X -0.006,Y -186.816,Z 1126.733,A 0.000,B 0.000,C 90.000,E1 131.881} C_DIS
LIN {X -0.060,Y -191.405,Z 1126.719,A 0.000,B 0.000,C 90.000,E1 129.402} C_DIS
LIN {X 0.021,Y -197.252,Z 1126.701,A 0.000,B 0.000,C 90.000,E1 126.091} C_DIS
LIN {X -0.021,Y -200.810,Z 1126.691,A 0.000,B 0.000,C 90.000,E1 124.326} C_DIS
LIN {X -0.067,Y -309.095,Z 1126.691,A 0.000,B 0.000,C 90.000,E1 124.326} C_DIS
LIN {X -0.011,Y -311.462,Z 1126.690,A 0.000,B 0.000,C 90.000,E1 124.278} C_DIS
LIN {X -0.134,Y -317.154,Z 1126.689,A 0.000,B 0.000,C 90.000,E1 123.992} C_DIS
LIN {X 0.008,Y -320.138,Z 1126.687,A 0.000,B 0.000,C 90.000,E1 123.658} C_DIS
LIN {X 0.006,Y -322.155,Z 1126.685,A 0.000,B 0.000,C 90.000,E1 123.372} C_DIS
LIN {X 0.002,Y -323.736,Z 1126.684,A 0.000,B 0.000,C 90.000,E1 123.086} C_DIS
LIN {X 0.091,Y -325.127,Z 1126.682,A 0.000,B 0.000,C 90.000,E1 122.752} C_DIS
LIN {X 0.029,Y -337.057,Z 1126.665,A 0.000,B 0.000,C 90.000,E1 119.617} C_DIS
LIN {X -0.163,Y -349.219,Z 1126.649,A 0.000,B 0.000,C 90.000,E1 116.873} C_DIS
LIN {X -0.020,Y -362.858,Z 1126.634,A 0.000,B 0.000,C 90.000,E1 114.131} C_DIS
LIN {X -0.040,Y -376.323,Z 1126.621,A 0.000,B 0.000,C 90.000,E1 111.770} C_DIS
LIN {X 0.005,Y -391.146,Z 1126.608,A 0.000,B 0.000,C 90.000,E1 109.450} C_DIS
LIN {X -0.210,Y -407.432,Z 1126.595,A 0.000,B 0.000,C 90.000,E1 107.221} C_DIS
LIN {X -0.150,Y -425.299,Z 1126.583,A 0.000,B 0.000,C 90.000,E1 105.009} C_DIS
LIN {X -0.200,Y -444.754,Z 1126.571,A 0.000,B 0.000,C 90.000,E1 102.883} C_DIS
LIN {X -0.098,Y -464.993,Z 1126.560,A 0.000,B 0.000,C 90.000,E1 100.894} C_DIS
LIN {X -0.070,Y -469.859,Z 1126.558,A 0.000,B 0.000,C 90.000,E1 100.423} C_DIS
LIN {X -0.121,Y -471.584,Z 1126.557,A 0.000,B 0.000,C 90.000,E1 100.197} C_DIS
LIN {X 0.200,Y -473.018,Z 1126.555,A 0.000,B 0.000,C 90.000,E1 99.905} C_DIS
LIN {X 0.055,Y -474.087,Z 1126.554,A 0.000,B 0.000,C 90.000,E1 99.670} C_DIS
LIN {X 0.170,Y -475.336,Z 1126.551,A 0.000,B 0.000,C 90.000,E1 99.151} C_DIS
LIN {X -0.103,Y -475.577,Z 1126.548,A 0.000,B 0.000,C 90.000,E1 98.681} C_DIS
LIN {X 0.026,Y -474.851,Z 1126.545,A 0.000,B 0.000,C 90.000,E1 98.163} C_DIS
LIN {X 0.160,Y -473.043,Z 1126.543,A 0.000,B 0.000,C 90.000,E1 97.644} C_DIS
LIN {X 0.022,Y -471.628,Z 1126.541,A 0.000,B 0.000,C 90.000,E1 97.409} C_DIS
LIN {X 0.142,Y -455.387,Z 1126.528,A 0.000,B 0.000,C 90.000,E1 95.106} C_DIS
LIN {X 0.072,Y -441.237,Z 1126.517,A 0.000,B 0.000,C 90.000,E1 93.037} C_DIS
LIN {X -0.213,Y -426.533,Z 1126.504,A 0.000,B 0.000,C 90.000,E1 90.688} C_DIS
LIN {X -0.024,Y -412.767,Z 1126.490,A 0.000,B 0.000,C 90.000,E1 88.224} C_DIS
LIN {X 0.060,Y -403.908,Z 1126.481,A 0.000,B 0.000,C 90.000,E1 86.560} C_DIS
LIN {X 0.015,Y -393.386,Z 1126.470,A 0.000,B 0.000,C 90.000,E1 84.609} C_DIS
LIN {X -0.170,Y -382.939,Z 1126.459,A 0.000,B 0.000,C 90.000,E1 82.648} C_DIS
LIN {X -0.090,Y -373.895,Z 1126.449,A 0.000,B 0.000,C 90.000,E1 80.905} C_DIS
LIN {X -0.158,Y -366.111,Z 1126.441,A 0.000,B 0.000,C 90.000,E1 79.454} C_DIS
LIN {X 0.038,Y -356.386,Z 1126.431,A 0.000,B 0.000,C 90.000,E1 77.645} C_DIS
LIN {X 0.133,Y -344.898,Z 1126.420,A 0.000,B 0.000,C 90.000,E1 75.519} C_DIS
LIN {X 0.087,Y -335.058,Z 1126.409,A 0.000,B 0.000,C 90.000,E1 73.685} C_DIS
LIN {X 0.065,Y -319.160,Z 1126.392,A 0.000,B 0.000,C 90.000,E1 70.550} C_DIS
LIN {X -0.104,Y -304.344,Z 1126.374,A 0.000,B 0.000,C 90.000,E1 67.358} C_DIS
LIN {X 0.039,Y -291.778,Z 1126.358,A 0.000,B 0.000,C 90.000,E1 64.357} C_DIS
LIN {X 0.078,Y -279.650,Z 1126.341,A 0.000,B 0.000,C 90.000,E1 61.307} C_DIS
LIN {X 0.125,Y -269.257,Z 1126.325,A 0.000,B 0.000,C 90.000,E1 58.535} C_DIS
LIN {X 0.050,Y -256.830,Z 1126.306,A 0.000,B 0.000,C 90.000,E1 55.022} C_DIS
LIN {X 0.025,Y -246.266,Z 1126.288,A 0.000,B 0.000,C 90.000,E1 51.778} C_DIS
LIN {X -0.056,Y -236.611,Z 1126.269,A 0.000,B 0.000,C 90.000,E1 48.485} C_DIS
LIN {X -0.038,Y -228.583,Z 1126.253,A 0.000,B 0.000,C 90.000,E1 45.486} C_DIS
LIN {X -0.050,Y -219.111,Z 1126.231,A 0.000,B 0.000,C 90.000,E1 41.676} C_DIS
LIN {X -0.132,Y -210.203,Z 1126.210,A 0.000,B 0.000,C 90.000,E1 37.810} C_DIS
LIN {X 0.089,Y -201.994,Z 1126.188,A 0.000,B 0.000,C 90.000,E1 33.785} C_DIS
LIN {X -0.003,Y -196.046,Z 1126.170,A 0.000,B 0.000,C 90.000,E1 30.590} C_DIS
LIN {X -0.026,Y -190.695,Z 1126.152,A 0.000,B 0.000,C 90.000,E1 27.334} C_DIS
LIN {X -0.007,Y -185.973,Z 1126.133,A 0.000,B 0.000,C 90.000,E1 24.027} C_DIS
LIN {X -0.056,Y -180.987,Z 1126.110,A 0.000,B 0.000,C 90.000,E1 19.866} C_DIS
LIN {X 0.059,Y -177.001,Z 1126.087,A 0.000,B 0.000,C 90.000,E1 15.607} C_DIS
LIN {X 0.002,Y -174.054,Z 1126.063,A 0.000,B 0.000,C 90.000,E1 11.366} C_DIS
LIN {X 0.077,Y -171.681,Z 1126.030,A 0.000,B 0.000,C 90.000,E1 5.334} C_DIS
LIN {X -0.038,Y -172.825,Z 1125.964,A 0.000,B 0.000,C 90.000,E1 353.514} C_DIS
LIN {X 0.044,Y -175.658,Z 1125.935,A 0.000,B 0.000,C 90.000,E1 348.342} C_DIS
LIN {X -0.018,Y -179.089,Z 1125.912,A 0.000,B 0.000,C 90.000,E1 344.102} C_DIS
LIN {X -0.026,Y -183.338,Z 1125.888,A 0.000,B 0.000,C 90.000,E1 339.880} C_DIS
LIN {X -0.051,Y -187.432,Z 1125.870,A 0.000,B 0.000,C 90.000,E1 336.538} C_DIS
LIN {X 0.001,Y -192.214,Z 1125.851,A 0.000,B 0.000,C 90.000,E1 333.204} C_DIS
LIN {X 0.009,Y -197.655,Z 1125.833,A 0.000,B 0.000,C 90.000,E1 329.921} C_DIS
LIN {X -0.090,Y -203.672,Z 1125.815,A 0.000,B 0.000,C 90.000,E1 326.707} C_DIS
LIN {X -0.048,Y -210.548,Z 1125.797,A 0.000,B 0.000,C 90.000,E1 323.497} C_DIS
LIN {X -0.086,Y -218.157,Z 1125.780,A 0.000,B 0.000,C 90.000,E1 320.356} C_DIS
LIN {X 0.048,Y -226.668,Z 1125.762,A 0.000,B 0.000,C 90.000,E1 317.229} C_DIS
LIN {X 0.064,Y -236.181,Z 1125.746,A 0.000,B 0.000,C 90.000,E1 314.190} C_DIS
LIN {X 0.023,Y -244.033,Z 1125.733,A 0.000,B 0.000,C 90.000,E1 311.962} C_DIS
LIN {X 0.018,Y -255.759,Z 1125.717,A 0.000,B 0.000,C 90.000,E1 309.036} C_DIS
LIN {X 0.048,Y -269.029,Z 1125.701,A 0.000,B 0.000,C 90.000,E1 306.171} C_DIS
LIN {X 0.078,Y -285.309,Z 1125.684,A 0.000,B 0.000,C 90.000,E1 303.038} C_DIS
LIN {X 0.097,Y -296.951,Z 1125.672,A 0.000,B 0.000,C 90.000,E1 301.003} C_DIS
LIN {X 0.015,Y -316.289,Z 1125.656,A 0.000,B 0.000,C 90.000,E1 298.052} C_DIS
LIN {X -0.167,Y -332.548,Z 1125.643,A 0.000,B 0.000,C 90.000,E1 295.848} C_DIS
LIN {X 0.150,Y -347.607,Z 1125.633,A 0.000,B 0.000,C 90.000,E1 293.951} C_DIS
LIN {X -0.047,Y -363.597,Z 1125.624,A 0.000,B 0.000,C 90.000,E1 292.259} C_DIS
LIN {X -0.002,Y -390.869,Z 1125.609,A 0.000,B 0.000,C 90.000,E1 289.704} C_DIS
LIN {X 0.120,Y -404.316,Z 1125.603,A 0.000,B 0.000,C 90.000,E1 288.489} C_DIS
LIN {X 0.129,Y -414.804,Z 1125.597,A 0.000,B 0.000,C 90.000,E1 287.511} C_DIS
LIN {X -0.223,Y -422.594,Z 1125.593,A 0.000,B 0.000,C 90.000,E1 286.804} C_DIS
LIN {X -0.181,Y -430.141,Z 1125.589,A 0.000,B 0.000,C 90.000,E1 286.024} C_DIS
LIN {X 0.160,Y -437.355,Z 1125.584,A 0.000,B 0.000,C 90.000,E1 285.190} C_DIS
LIN {X 0.018,Y -444.169,Z 1125.580,A 0.000,B 0.000,C 90.000,E1 284.411} C_DIS
LIN {X -0.175,Y -450.383,Z 1125.576,A 0.000,B 0.000,C 90.000,E1 283.647} C_DIS
LIN {X 0.125,Y -455.943,Z 1125.571,A 0.000,B 0.000,C 90.000,E1 282.827} C_DIS
LIN {X 0.040,Y -460.709,Z 1125.567,A 0.000,B 0.000,C 90.000,E1 282.063} C_DIS
LIN {X -0.013,Y -464.856,Z 1125.563,A 0.000,B 0.000,C 90.000,E1 281.299} C_DIS
LIN {X -0.115,Y -468.491,Z 1125.558,A 0.000,B 0.000,C 90.000,E1 280.546} C_DIS
LIN {X -0.185,Y -471.587,Z 1125.554,A 0.000,B 0.000,C 90.000,E1 279.792} C_DIS
LIN {X -0.012,Y -473.343,Z 1125.552,A 0.000,B 0.000,C 90.000,E1 279.265} C_DIS
LIN {X 0.097,Y -474.796,Z 1125.549,A 0.000,B 0.000,C 90.000,E1 278.746} C_DIS
LIN {X -0.184,Y -475.960,Z 1125.546,A 0.000,B 0.000,C 90.000,E1 278.276} C_DIS
LIN {X -0.055,Y -476.858,Z 1125.543,A 0.000,B 0.000,C 90.000,E1 277.757} C_DIS
LIN {X 0.082,Y -477.430,Z 1125.540,A 0.000,B 0.000,C 90.000,E1 277.239} C_DIS
LIN {X 0.226,Y -477.694,Z 1125.537,A 0.000,B 0.000,C 90.000,E1 276.720} C_DIS
LIN {X -0.101,Y -477.626,Z 1125.535,A 0.000,B 0.000,C 90.000,E1 276.258} C_DIS
LIN {X 0.048,Y -477.223,Z 1125.532,A 0.000,B 0.000,C 90.000,E1 275.739} C_DIS
LIN {X 0.194,Y -476.540,Z 1125.529,A 0.000,B 0.000,C 90.000,E1 275.220} C_DIS
LIN {X -0.137,Y -475.453,Z 1125.526,A 0.000,B 0.000,C 90.000,E1 274.759} C_DIS
LIN {X -0.036,Y -473.988,Z 1125.524,A 0.000,B 0.000,C 90.000,E1 274.245} C_DIS
LIN {X 0.095,Y -471.973,Z 1125.521,A 0.000,B 0.000,C 90.000,E1 273.726} C_DIS
LIN {X -0.094,Y -470.775,Z 1125.519,A 0.000,B 0.000,C 90.000,E1 273.498} C_DIS
LIN {X 0.015,Y -467.698,Z 1125.517,A 0.000,B 0.000,C 90.000,E1 272.980} C_DIS
LIN {X -0.181,Y -465.848,Z 1125.515,A 0.000,B 0.000,C 90.000,E1 272.751} C_DIS
LIN {X -0.121,Y -461.289,Z 1125.512,A 0.000,B 0.000,C 90.000,E1 272.236} C_DIS
LIN {X 0.128,Y -458.497,Z 1125.511,A 0.000,B 0.000,C 90.000,E1 271.949} C_DIS
LIN {X -0.067,Y -455.318,Z 1125.510,A 0.000,B 0.000,C 90.000,E1 271.718} C_DIS
LIN {X 0.130,Y -448.840,Z 1125.507,A 0.000,B 0.000,C 90.000,E1 271.260} C_DIS
LIN {X -0.023,Y -442.084,Z 1125.505,A 0.000,B 0.000,C 90.000,E1 270.917} C_DIS
LIN {X -0.160,Y -435.059,Z 1125.503,A 0.000,B 0.000,C 90.000,E1 270.630} C_DIS
LIN {X 0.077,Y -427.992,Z 1125.502,A 0.000,B 0.000,C 90.000,E1 270.344} C_DIS
LIN {X 0.191,Y -420.800,Z 1125.501,A 0.000,B 0.000,C 90.000,E1 270.115} C_DIS
LIN {X 0.147,Y -413.457,Z 1125.500,A 0.000,B 0.000,C 90.000,E1 269.943} C_DIS
LIN {X -0.076,Y -402.167,Z 1125.499,A 0.000,B 0.000,C 90.000,E1 269.771} C_DIS
LIN {X 0.007,Y -392.454,Z 1125.498,A 0.000,B 0.000,C 90.000,E1 269.656} C_DIS
LIN {X 0.092,Y -382.543,Z 1125.498,A 0.000,B 0.000,C 90.000,E1 269.599} C_DIS
LIN {X 0.022,Y -181.466,Z 1125.498,A 0.000,B 0.000,C 90.000,E1 269.599} C_DIS
LIN {X -0.023,Y -180.906,Z 1125.474,A 0.000,B 0.000,C 90.000,E1 265.355} C_DIS
LIN {X 0.050,Y -180.678,Z 1125.469,A 0.000,B 0.000,C 90.000,E1 264.489} C_DIS
LIN {X -0.051,Y -178.761,Z 1125.441,A 0.000,B 0.000,C 90.000,E1 259.454} C_DIS
LIN {X 0.021,Y -175.807,Z 1125.413,A 0.000,B 0.000,C 90.000,E1 254.338} C_DIS
LIN {X 0.015,Y -171.993,Z 1125.385,A 0.000,B 0.000,C 90.000,E1 249.209} C_DIS
LIN {X 0.053,Y -171.404,Z 1125.380,A 0.000,B 0.000,C 90.000,E1 248.337} C_DIS
LIN {X 0.038,Y -167.645,Z 1125.356,A 0.000,B 0.000,C 90.000,E1 244.024} C_DIS
LIN {X 0.052,Y -166.308,Z 1125.346,A 0.000,B 0.000,C 90.000,E1 242.281} C_DIS
LIN {X 0.047,Y -163.051,Z 1125.327,A 0.000,B 0.000,C 90.000,E1 238.791} C_DIS
LIN {X 0.008,Y -160.985,Z 1125.312,A 0.000,B 0.000,C 90.000,E1 236.167} C_DIS
LIN {X -0.015,Y -157.734,Z 1125.292,A 0.000,B 0.000,C 90.000,E1 232.637} C_DIS
LIN {X -0.076,Y -155.773,Z 1125.278,A 0.000,B 0.000,C 90.000,E1 229.989} C_DIS
LIN {X -0.020,Y -152.028,Z 1125.253,A 0.000,B 0.000,C 90.000,E1 225.486} C_DIS
LIN {X -0.003,Y -150.275,Z 1125.238,A 0.000,B 0.000,C 90.000,E1 222.771} C_DIS
LIN {X 0.015,Y -147.026,Z 1125.212,A 0.000,B 0.000,C 90.000,E1 218.222} C_DIS
LIN {X 0.035,Y -145.608,Z 1125.197,A 0.000,B 0.000,C 90.000,E1 215.471} C_DIS
LIN {X 0.040,Y -142.993,Z 1125.172,A 0.000,B 0.000,C 90.000,E1 210.875} C_DIS
LIN {X -0.025,Y -141.621,Z 1125.151,A 0.000,B 0.000,C 90.000,E1 207.206} C_DIS
LIN {X 0.030,Y -139.431,Z 1125.115,A 0.000,B 0.000,C 90.000,E1 200.684} C_DIS
LIN {X -0.046,Y -139.162,Z 1125.105,A 0.000,B 0.000,C 90.000,E1 198.852} C_DIS
LIN {X -0.009,Y -138.341,Z 1125.058,A 0.000,B 0.000,C 90.000,E1 190.433} C_DIS
LIN {X -0.001,Y -139.479,Z 1125.006,A 0.000,B 0.000,C 90.000,E1 181.088} C_DIS
LIN {X -0.061,Y -141.065,Z 1124.975,A 0.000,B 0.000,C 90.000,E1 175.527} C_DIS
LIN {X 0.034,Y -142.440,Z 1124.960,A 0.000,B 0.000,C 90.000,E1 172.704} C_DIS
LIN {X -0.046,Y -144.678,Z 1124.934,A 0.000,B 0.000,C 90.000,E1 168.117} C_DIS
